FUNCTION_BLOCK FB 1001
TITLE = HOPPER
//Creation:
//Date:            Author:                                               Version
//-------------------------------------------------------------------------------
//-
//17.10.19          Ilia Bedniakov (ilia   )                             01.00.00
//
//Changes:
//No. Date:        Who       Description                           Mark   Version 
//-------------------------------------------------------------------------------
//- 
//               
//_______________________________________________________________________________
//_
//Function:
AUTHOR : ilia
NAME : project
VERSION : 0.1
VAR_INPUT
  i_xSystemActive : BOOL ;	//system control on
  i_xFAValveOpen : BOOL ;
  i_xFAValveClosed : BOOL ;
  i_xPBStart : BOOL ;	//Start Button
  i_xPBStop : BOOL ;	//StopButton
  i_xCstAvailable : BOOL ;	//Container On Place
  ack_FAValve : BOOL ;	//acknowlege FAValve
END_VAR
VAR_IN_OUT
  q_xFAValve : BOOL ;	//Open Fresh Air Valve
  q_xPFCMix : BOOL ;	//Container in position PFC to MIX01
  q_xLMStart : BOOL ;
  q_xLMCstAvalible : BOOL ;
  f_xFAValve : BOOL ;	//feedback fault
END_VAR
VAR
  reserve_IO : ARRAY  [4 .. 49 ] OF BYTE ;
  HMI : STRUCT 	//Interface of HMI
   CMD : STRUCT
    xxRes1 : BOOL ;
    xSetEmpty : BOOL ;
    xStopBtnTest : BOOL ;
    xStartBtnTest : BOOL ;
    xContainerPlaceTest : BOOL ;
    reserve_5 : BOOL ;
    reserve_6 : BOOL ;
    reserve_7 : BOOL ;
    reserve_8 : BOOL ;
    reserve_9 : BOOL ;
    reserve_10 : BOOL ;
    reserve_11 : BOOL ;
    reserve_12 : BOOL ;
    reserve_13 : BOOL ;
    reserve_14 : BOOL ;
    reserve_15 : BOOL ;
   END_STRUCT ;
   STATE : STRUCT
    xFaulted : BOOL ;
    xContainer : BOOL ;
    reserve_2 : BOOL ;
    reserve_3 : BOOL ;
    reserve_4 : BOOL ;
    xFilled : BOOL ;
    xEmpty : BOOL ;
    reserve_7 : BOOL ;
    reserve_8 : BOOL ;
    reserve_9 : BOOL ;
    reserve_10 : BOOL ;
    reserve_11 : BOOL ;
    reserve_12 : BOOL ;
    reserve_13 : BOOL ;
    reserve_14 : BOOL ;
    reserve_15 : BOOL ;
   END_STRUCT ;
   PARAM : STRUCT
    rDischargeTime : REAL  := 2.000000e+000;
    reserve_1 : REAL  := 6.000000e+001;
    reserve_2 : REAL  := 6.000000e+001;
    reserve_3 : REAL  := 6.000000e+001;
    reserve_4 : REAL ;
    reserve_5 : REAL ;
    reserve_6 : REAL ;
    reserve_7 : REAL ;
    reserve_8 : INT ;
    reserve_9 : INT ;
    reserve_10 : INT ;
    reserve_11 : INT ;
    reserve_12 : INT ;
    reserve_14 : INT ;
    reserve_15 : INT ;
   END_STRUCT ;
   PV : STRUCT
    rDischargeTime : REAL ;	//Minutes
    reserve_1_4 : REAL  := 6.000000e+001;
    reserve_2 : REAL  := 6.000000e+001;
    reserve_3 : REAL  := 6.000000e+001;
    reserve_4 : REAL ;
    reserve_5 : REAL ;
    reserve_6 : REAL ;
    reserve_7 : REAL ;
    iRecipeNumber : INT ;
    reserve_9 : INT ;
    reserve_10 : INT ;
    reserve_11 : INT ;
    reserve_12 : INT ;
    reserve_14 : INT ;
    reserve_15 : INT ;
   END_STRUCT ;
  END_STRUCT ;
  reserve_HMI : ARRAY  [146 .. 199 ] OF BYTE ;
  PROD : STRUCT 	//Interface of Production
   FROM : STRUCT
    reserve : INT ;
    reserve_1 : INT ;
    reserve_2 : INT ;
    reserve_3 : INT ;
    reserve_4 : INT ;
    reserve_5 : REAL ;
    reserve_6 : REAL ;
    CMD : STRUCT
     reserve : BOOL ;
     reserve_1 : BOOL ;
     reserve_2 : BOOL ;
     reserve_3 : BOOL ;
     reserve_4 : BOOL ;
     reserve_5 : BOOL ;
     reserve_6 : BOOL ;
     reserve_7 : BOOL ;
     reserve_8 : BOOL ;
     reserve_9 : BOOL ;
     reserve_10 : BOOL ;
     reserve_11 : BOOL ;
     reserve_12 : BOOL ;
     reserve_13 : BOOL ;
     reserve_14 : BOOL ;
     reserve_15 : BOOL ;
    END_STRUCT ;
   END_STRUCT ;
   TO : STRUCT
    reserve : INT ;
    reserve_1 : INT ;
    reserve_2 : INT ;
    reserve_3 : INT ;
    reserve_4 : INT ;
    reserve_5 : REAL ;
    reserve_6 : REAL ;
    STATE : STRUCT
     reserve : BOOL ;
     reserve_1 : BOOL ;
     reserve_2 : BOOL ;
     reserve_3 : BOOL ;
     reserve_4 : BOOL ;
     reserve_5 : BOOL ;
     reserve_6 : BOOL ;
     reserve_7 : BOOL ;
     reserve_8 : BOOL ;
     reserve_9 : BOOL ;
     reserve_10 : BOOL ;
     reserve_11 : BOOL ;
     reserve_12 : BOOL ;
     reserve_13 : BOOL ;
     reserve_14 : BOOL ;
     reserve_15 : BOOL ;
    END_STRUCT ;
   END_STRUCT ;
   reserve : ARRAY  [40 .. 49 ] OF BYTE ;
  END_STRUCT ;
  IF_CONSUMER : STRUCT 	//Interface scale in storage location
   CONTROL : STRUCT
    Answer_DB : INT ;
    Answer_DW : INT ;
    iRecipeNumber : INT ;
    rRes1 : REAL ;
    iPulseValve : REAL ;
    iPauseValve : REAL ;
    CMD : STRUCT
     xConnect : BOOL ;
     xRequest : BOOL ;
     xRelease : BOOL ;
     xFull : BOOL ;
     xCleaningRelease : BOOL ;
     xPressureFault : BOOL ;
     xAckRecipe : BOOL ;
     xPulseCondition : BOOL ;
     xDischargeActive : BOOL ;
     reserve_9 : BOOL ;
     reserve_10 : BOOL ;
     reserve_11 : BOOL ;
     reserve_12 : BOOL ;
     reserve_13 : BOOL ;
     reserve_14 : BOOL ;
     reserve_15 : BOOL ;
    END_STRUCT ;
   END_STRUCT ;
   STATUS : STRUCT
    reserve_1 : INT ;
    reserve_2 : INT ;
    iRecipeNumber : INT ;
    rRes1 : REAL ;
    rRes2 : REAL ;
    rRes3 : REAL ;
    STATE : STRUCT
     xReady : BOOL ;
     xActive : BOOL ;
     xStopped : BOOL ;
     xStarted : BOOL ;
     xEmpty : BOOL ;
     reserve_5 : BOOL ;
     reserve_6 : BOOL ;
     reserve_7 : BOOL ;
     reserve_8 : BOOL ;
     reserve_9 : BOOL ;
     reserve_10 : BOOL ;
     reserve_11 : BOOL ;
     reserve_12 : BOOL ;
     reserve_13 : BOOL ;
     reserve_14 : BOOL ;
     reserve_15 : BOOL ;
    END_STRUCT ;
   END_STRUCT ;
  END_STRUCT ;
  reserve_IF : ARRAY  [290 .. 499 ] OF BYTE ;
  FAValve : STRUCT 	//valve object with 1Q and 0-2I
   parameter : STRUCT
    valve_on : BOOL  := TRUE;	//activate valve structure
    clock_on : BOOL  := TRUE;	//activate clock structure
    reserve_3 : BOOL ;
    switching_number_on : BOOL ;	//activate switching number counter
    reserve_4 : BOOL ;
    parameter_1Q : BOOL ;	//valve type with 1 quit 0 inputs
    parameter_1Q_1I : BOOL ;	//valve type with 1 quit 1 input (=)
    parameter_1Q_1IN : BOOL ;	//valve type with 1 quit 1 input (<>)
    parameter_1Q_2I : BOOL  := TRUE;	//valve type with 1 quit 2 inputs
    parameter_text_pos_1 : BOOL ;
    parameter_text_straight : BOOL ;
    parameter_text_inverse : BOOL  := TRUE;	//select text inverse = "close/open" or "bypass/convey" aso.
    parameter_text_open : BOOL  := TRUE;	//select text quit = "open/close"
    parameter_text_convey : BOOL ;	//select text quit = "convey/bypass"
    parameter_text_on : BOOL ;	//select text quit = "on/off"
    parameter_text_up : BOOL ;	//select text quit = "up/down"
   END_STRUCT ;
   quit_valve : BOOL ;	//1 = quit valve
   input_valve_set : BOOL ;	//1 = input valve, if quit valve set
   input_valve_not_set : BOOL ;	//1 = input valve, if quit valve not set
   auto_mode_control : BOOL ;	//1 = release/control of valve in auto mode
   valve_in_operation : BOOL ;	//1 = signal valve in operation
   fault : BOOL ;	//1 = signal valve fault
   man_mode_to_SCADA : BOOL ;	//0 = automatic mode , 1 = manual mode
   man_mode_from_SCADA : BOOL ;	//0 = automatic mode , 1 = manual mode
   man_mode_control : BOOL ;	//1 = release/control of valve in manual mode (from SCADA)
   man_mode_locked : BOOL ;	//1 = change to manual mode locked, valve is in automatic use
   start_with_impulse : BOOL  := TRUE;	//1 = start cycle with impluse
   set_cycles_reached : BOOL ;	//1 = set number of cycles has been reached
   continous_clock : BOOL  := TRUE;	//1 = continous clock / 0 = set number of clocks
   simulation : BOOL ;	//1 = simulation of object
   release_clock : BOOL  := TRUE;	//1 = release bit for clock FC
   quit_clock : BOOL ;	//quit for clock FC, if release_clock = TRUE
   set_time_fault : INT  := 5;	//fault evaluation time in seconds
   actual_time_fault : INT ;	//actual fault evaluation time in seconds
   impulse_time : REAL  := 5.000000e+000;	//impulse time for clock in seconds
   break_time : REAL  := 5.000000e+000;	//break time for clock in seconds
   time_counter : REAL ;	//time counter (elapsed time)
   set_cycles : INT ;	//number of clocks if not continous clock
   clock_counter : INT ;	//clock counter
   switching_number_counter : STRUCT 	//switching number counter
    reset : BOOL ;	//reset switching number counter
    warning : BOOL ;	//warning number exceeded
    alarm : BOOL ;	//alarm number exceeded
    flank_flag : BOOL ;	//internal flag
    actual_switching_number : REAL ;	//actual switching number
    set_number_warning : REAL ;	//set number for warning
    set_number_alarm : REAL ;	//set number for alarm
   END_STRUCT ;
   set_time_in_operation : INT ;	//1IoO: set time for delay of "valve in operation"
   real_time_in_operation : INT ;	//1IoO: real time for delay of "valve in operation"
   system_on : BOOL ;	//system released resepectively system area released after emergency stopping
   reserve : ARRAY  [44 .. 47 ] OF BYTE ;
   object_state : INT ;	//1=grey; 5=green; 9=white; 15=yellow; 16=red
  END_STRUCT ;
  reserve_Cmod_1 : ARRAY  [550 .. 799 ] OF BYTE ;
  BinaryObjects : STRUCT
   PBStart : STRUCT
    parameter : STRUCT
     reserve : BOOL ;
     debounce_time : BOOL ;	//view/edit debounce time
     reserve_2 : BOOL ;
     switching_number_counter : BOOL ;	//Counter for operating cycles
     reserve_4 : BOOL ;
     reserve_5 : BOOL ;
     reserve_6 : BOOL ;
     reserve_7 : BOOL ;
     parameter_invers : BOOL ;	//Parameter signal invers, invert the status
     reserve_9 : BOOL ;
     reserve_10 : BOOL ;
     reserve_11 : BOOL ;
     reserve_12 : BOOL ;
     reserve_13 : BOOL ;
     reserve_14 : BOOL ;
     reserve_15 : BOOL ;
    END_STRUCT ;
    input_processed : BOOL ;	//Input_signal processed
    input : BOOL ;	//Input signal
    def_invert_input : BOOL ;	//Definition to invert input signal (1=invert input)
    def_debounce_input : BOOL ;	//Definition to debounce input signal (1=debounce input)
    def_fault_state : BOOL ;	//Definition of fault state
    fault : BOOL ;	//1 = fault message
    man_mode_to_SCADA : BOOL ;	//0=Automode; 1=Manualmode
    man_mode_from_SCADA : BOOL ;	//0=Automode; 1=Manualmode
    man_mode_control : BOOL ;	//Control the object in manual mode (from scada)
    man_mode_locked : BOOL ;	//Lock manual mode, because object is used in auto mode
    system_on : BOOL ;
    spare : BOOL ;
    input_inverted : BOOL ;	//Input signal inverted if necessary
    input_debounced : BOOL ;	//Input signal debounced if necessary (also inverted if necessary9)
    input_debounced_high : BOOL ;	//Input signal debounced high (output signal timer)
    input_debounced_low : BOOL ;	//Input signal debounced low (output signal timer)
    set_time_fault : INT ;	//Set value fault evaulation time
    act_time_fault : INT ;	//Act value fault avaulation time
    set_time_debounced_high : REAL ;
    act_time_debounced_high : REAL ;
    set_time_debounced_low : REAL ;
    act_time_debounced_low : REAL ;
    cycle_counter : STRUCT
     reset_counter : BOOL ;	//Reset operating cycle counter
     warning : BOOL ;	//Warning time 1 elapsed
     alarm : BOOL ;	//Alarm time 2 elapsed
     flank_flag : BOOL ;	//Intern used flag
     act_number_of_cycles : REAL ;	//Actual number of cycles (cycle counter)
     set_number_warning : REAL ;	//Set value for generate the warning
     set_number_alarm : REAL ;	//Set value for generate the alarm
    END_STRUCT ;
    reserve : ARRAY  [38 .. 47 ] OF BYTE ;
    object_state : INT ;
   END_STRUCT ;
   PBStop : STRUCT
    parameter : STRUCT
     reserve : BOOL ;
     debounce_time : BOOL ;	//view/edit debounce time
     reserve_2 : BOOL ;
     switching_number_counter : BOOL ;	//Counter for operating cycles
     reserve_4 : BOOL ;
     reserve_5 : BOOL ;
     reserve_6 : BOOL ;
     reserve_7 : BOOL ;
     parameter_invers : BOOL ;	//Parameter signal invers, invert the status
     reserve_9 : BOOL ;
     reserve_10 : BOOL ;
     reserve_11 : BOOL ;
     reserve_12 : BOOL ;
     reserve_13 : BOOL ;
     reserve_14 : BOOL ;
     reserve_15 : BOOL ;
    END_STRUCT ;
    input_processed : BOOL ;	//Input_signal processed
    input : BOOL ;	//Input signal
    def_invert_input : BOOL ;	//Definition to invert input signal (1=invert input)
    def_debounce_input : BOOL ;	//Definition to debounce input signal (1=debounce input)
    def_fault_state : BOOL ;	//Definition of fault state
    fault : BOOL ;	//1 = fault message
    man_mode_to_SCADA : BOOL ;	//0=Automode; 1=Manualmode
    man_mode_from_SCADA : BOOL ;	//0=Automode; 1=Manualmode
    man_mode_control : BOOL ;	//Control the object in manual mode (from scada)
    man_mode_locked : BOOL ;	//Lock manual mode, because object is used in auto mode
    system_on : BOOL ;
    spare : BOOL ;
    input_inverted : BOOL ;	//Input signal inverted if necessary
    input_debounced : BOOL ;	//Input signal debounced if necessary (also inverted if necessary9)
    input_debounced_high : BOOL ;	//Input signal debounced high (output signal timer)
    input_debounced_low : BOOL ;	//Input signal debounced low (output signal timer)
    set_time_fault : INT ;	//Set value fault evaulation time
    act_time_fault : INT ;	//Act value fault avaulation time
    set_time_debounced_high : REAL ;
    act_time_debounced_high : REAL ;
    set_time_debounced_low : REAL ;
    act_time_debounced_low : REAL ;
    cycle_counter : STRUCT
     reset_counter : BOOL ;	//Reset operating cycle counter
     warning : BOOL ;	//Warning time 1 elapsed
     alarm : BOOL ;	//Alarm time 2 elapsed
     flank_flag : BOOL ;	//Intern used flag
     act_number_of_cycles : REAL ;	//Actual number of cycles (cycle counter)
     set_number_warning : REAL ;	//Set value for generate the warning
     set_number_alarm : REAL ;	//Set value for generate the alarm
    END_STRUCT ;
    reserve : ARRAY  [38 .. 47 ] OF BYTE ;
    object_state : INT ;
   END_STRUCT ;
   PBCstAvailable : STRUCT
    parameter : STRUCT
     reserve : BOOL ;
     debounce_time : BOOL ;	//view/edit debounce time
     reserve_2 : BOOL ;
     switching_number_counter : BOOL ;	//Counter for operating cycles
     reserve_4 : BOOL ;
     reserve_5 : BOOL ;
     reserve_6 : BOOL ;
     reserve_7 : BOOL ;
     parameter_invers : BOOL ;	//Parameter signal invers, invert the status
     reserve_9 : BOOL ;
     reserve_10 : BOOL ;
     reserve_11 : BOOL ;
     reserve_12 : BOOL ;
     reserve_13 : BOOL ;
     reserve_14 : BOOL ;
     reserve_15 : BOOL ;
    END_STRUCT ;
    input_processed : BOOL ;	//Input_signal processed
    input : BOOL ;	//Input signal
    def_invert_input : BOOL ;	//Definition to invert input signal (1=invert input)
    def_debounce_input : BOOL ;	//Definition to debounce input signal (1=debounce input)
    def_fault_state : BOOL ;	//Definition of fault state
    fault : BOOL ;	//1 = fault message
    man_mode_to_SCADA : BOOL ;	//0=Automode; 1=Manualmode
    man_mode_from_SCADA : BOOL ;	//0=Automode; 1=Manualmode
    man_mode_control : BOOL ;	//Control the object in manual mode (from scada)
    man_mode_locked : BOOL ;	//Lock manual mode, because object is used in auto mode
    system_on : BOOL ;
    spare : BOOL ;
    input_inverted : BOOL ;	//Input signal inverted if necessary
    input_debounced : BOOL ;	//Input signal debounced if necessary (also inverted if necessary9)
    input_debounced_high : BOOL ;	//Input signal debounced high (output signal timer)
    input_debounced_low : BOOL ;	//Input signal debounced low (output signal timer)
    set_time_fault : INT ;	//Set value fault evaulation time
    act_time_fault : INT ;	//Act value fault avaulation time
    set_time_debounced_high : REAL ;
    act_time_debounced_high : REAL ;
    set_time_debounced_low : REAL ;
    act_time_debounced_low : REAL ;
    cycle_counter : STRUCT
     reset_counter : BOOL ;	//Reset operating cycle counter
     warning : BOOL ;	//Warning time 1 elapsed
     alarm : BOOL ;	//Alarm time 2 elapsed
     flank_flag : BOOL ;	//Intern used flag
     act_number_of_cycles : REAL ;	//Actual number of cycles (cycle counter)
     set_number_warning : REAL ;	//Set value for generate the warning
     set_number_alarm : REAL ;	//Set value for generate the alarm
    END_STRUCT ;
    reserve : ARRAY  [38 .. 47 ] OF BYTE ;
    object_state : INT ;
   END_STRUCT ;
  END_STRUCT ;
  reserve_Cmod : ARRAY  [950 .. 1499 ] OF BYTE ;
  TIMES : STRUCT 	//ten timers
   TON_VibroRinneFault : STRUCT
    IN : BOOL ;
    RST : BOOL ;
    IMP : BOOL ;
    Q : BOOL ;
    PT : REAL ;
    ET : REAL ;
   END_STRUCT ;
   TON_Restdischarge : STRUCT
    IN : BOOL ;
    RST : BOOL ;
    IMP : BOOL ;
    Q : BOOL ;
    PT : REAL ;
    ET : REAL ;
   END_STRUCT ;
   TON_VibroRinneStart : STRUCT
    IN : BOOL ;
    RST : BOOL ;
    IMP : BOOL ;
    Q : BOOL ;
    PT : REAL ;
    ET : REAL ;
   END_STRUCT ;
   TON_HopperDischarge : STRUCT
    IN : BOOL ;
    RST : BOOL ;
    IMP : BOOL ;
    Q : BOOL ;
    PT : REAL ;
    ET : REAL ;
   END_STRUCT ;
   TON_Vibrorinne : STRUCT
    IN : BOOL ;
    RST : BOOL ;
    IMP : BOOL ;
    Q : BOOL ;
    PT : REAL ;
    ET : REAL ;
   END_STRUCT ;
  END_STRUCT ;
  SEQUENCES : STRUCT
   Filling : STRUCT
    AUTO : BOOL ;
    MANUAL : BOOL ;
    LOCKED : BOOL ;
    reserve : BOOL ;
    reserve_1 : BOOL ;
    reserve_2 : BOOL ;
    reserve_3 : BOOL ;
    reserve_4 : BOOL ;
    reserve_5 : BOOL ;
    reserve_6 : BOOL ;
    reserve_7 : BOOL ;
    reserve_8 : BOOL ;
    reserve_9 : BOOL ;
    reserve_10 : BOOL ;
    reserve_11 : BOOL ;
    reserve_12 : BOOL ;
   END_STRUCT ;
   Discharging : STRUCT
    AUTO : BOOL ;
    MANUAL : BOOL ;
    LOCKED : BOOL ;
    RELEASED : BOOL ;
    ACTIVE : BOOL ;
    HOPPERDISCHARGE : BOOL ;
    FAULTED : BOOL ;
    CLEANING : BOOL ;
    reserve_5 : BOOL ;
    reserve_6 : BOOL ;
    reserve_7 : BOOL ;
    reserve_8 : BOOL ;
    reserve_9 : BOOL ;
    reserve_10 : BOOL ;
    reserve_11 : BOOL ;
    reserve_15 : BOOL ;
   END_STRUCT ;
   reserve : ARRAY  [4 .. 99 ] OF BYTE ;
  END_STRUCT ;
  INTERNAL : STRUCT
   IF : STRUCT
    RECEIVER : STRUCT
     res : BOOL ;
     res_1 : BOOL ;
     res_2 : BOOL ;
     res_3 : BOOL ;
     res_4 : BOOL ;
     res_5 : BOOL ;
     res_6 : BOOL ;
     res_7 : BOOL ;
    END_STRUCT ;
    reserve_1 : BOOL ;
    reserve_2 : BOOL ;
    reserve_3 : BOOL ;
    reserve_4 : BOOL ;
    reserve_5 : BOOL ;
    reserve_6 : BOOL ;
    reserve_7 : BOOL ;
    reserve_8 : BOOL ;
    reserve_9 : BOOL ;
    reserve_10 : BOOL ;
    reserve_11 : BOOL ;
    reserve_12 : BOOL ;
    reserve_13 : BOOL ;
    reserve_14 : BOOL ;
    reserve_14_1 : BOOL ;
   END_STRUCT ;
   Flags : STRUCT
    FP_start : STRUCT
     helpbit : BOOL ;
     pulsebit : BOOL ;
    END_STRUCT ;
    FN_cleaning : STRUCT
     helpbit : BOOL ;
     pulsebit : BOOL ;
    END_STRUCT ;
    res_2 : BOOL ;
    res_3 : BOOL ;
    res_2_1 : BOOL ;
    res_3_1 : BOOL ;
    res_3_1_1 : BOOL ;
   END_STRUCT ;
   CSTStatus : STRUCT
    xx_xFull : BOOL ;
    xFilled : BOOL ;
    xEmptyOrDischarged : BOOL ;
    xCSTAvailable : BOOL ;
    xCleanedPipe : BOOL ;
    reserve_5 : BOOL ;
    reserve_6 : BOOL ;
    reserve_7 : BOOL ;
    xValveExtraCond : BOOL ;
   END_STRUCT ;
   CSTProcessStatus : STRUCT
    xStartCMDActive : BOOL ;
    reserve_1 : BOOL ;
    reserve_2 : BOOL ;
    reserve_3 : BOOL ;
    reserve_4 : BOOL ;
    reserve_5 : BOOL ;
    reserve_6 : BOOL ;
    reserve_7 : BOOL ;
   END_STRUCT ;
   Switches : STRUCT
    res1 : BOOL ;
    res2 : BOOL ;
    res3 : BOOL ;
    res4 : BOOL ;
    res5 : BOOL ;
    res6 : BOOL ;
    res7 : BOOL ;
    ress8 : BOOL ;
    res9 : BOOL ;
    res10 : BOOL ;
    res11 : BOOL ;
   END_STRUCT ;
   BUTTONS_LAMPS : STRUCT
    LMStart : STRUCT
     Steady : BOOL ;
     Flash : BOOL ;
     DoubleFlash : BOOL ;
     Activated : BOOL ;
     res_1 : BOOL ;
     res_2 : BOOL ;
     res_3 : BOOL ;
     res_4 : BOOL ;
    END_STRUCT ;
    LMStop : STRUCT
     Steady : BOOL ;
     Flash : BOOL ;
     DoubleFlash : BOOL ;
     Activated : BOOL ;
     res_1 : BOOL ;
     res_2 : BOOL ;
     res_3 : BOOL ;
     res_4 : BOOL ;
    END_STRUCT ;
    LMCstAvailable : STRUCT
     Steady : BOOL ;
     Flash : BOOL ;
     DoubleFlash : BOOL ;
     Activated : BOOL ;
     res_1 : BOOL ;
     res_2 : BOOL ;
     res_3 : BOOL ;
     res_4 : BOOL ;
    END_STRUCT ;
    res_2_2 : BOOL ;
    res_3 : BOOL ;
    res_4 : BOOL ;
    res_5 : BOOL ;
    res_1_1 : BOOL ;
    res_2_1 : BOOL ;
    res_3_1 : BOOL ;
    res_4_1 : BOOL ;
    res_1 : BOOL ;
    res_2 : BOOL ;
   END_STRUCT ;
   Instance_DB_number : INT ;
  END_STRUCT ;
END_VAR
VAR_TEMP
  tempREAL : REAL ;
  tempINT : INT ;
  tempWORD : WORD ;
  tempBOOL : BOOL ;
END_VAR
BEGIN
NETWORK
TITLE = ------------------ INSTANCE DB (STANDART)-----------------------
      L     0;
      L     DINO;
      ==I;
      BEC;
      T     #INTERNAL.Instance_DB_number;
NETWORK
TITLE = -------------SEQUENCES AUTO/LOCKED/MANUAL-----------------
NETWORK
TITLE = Sequence discharging auto
      A     #IF_CONSUMER.CONTROL.CMD.xRequest;
      AN    #SEQUENCES.Discharging.LOCKED;
      =     #SEQUENCES.Discharging.AUTO;
NETWORK
TITLE = Sequence discharging manual
      O     #FAValve.man_mode_to_SCADA;
      =     #SEQUENCES.Discharging.MANUAL;
NETWORK
TITLE = Sequence discharging locked
      O     #SEQUENCES.Discharging.MANUAL;
      ON    #i_xSystemActive;
      =     #SEQUENCES.Discharging.LOCKED;
NETWORK
TITLE = ------------- SENSORS/SWITCHES/BINARY --------------------------
NETWORK
TITLE = LMP PBStart
      O     #i_xPBStart;
      O     #HMI.CMD.xStartBtnTest;
      =     #i_xPBStart;
      CALL  FC 24 (
           in_Handbedienung_erlaubt := TRUE,
           in_Anlage_ein            := #i_xSystemActive,
           in_Eingang               := #i_xPBStart,
           in_Eingang_drehen        := FALSE,
           in_Eingang_entprellen    := FALSE,
           in_Stoerauswertung_aktiv := FALSE,
           in_Quitt_Stoerung_noetig := FALSE,
           in_Stoer_Zustand         := FALSE,
           in_Quitt_Stoerung        := FALSE,
           io_Eingang_verarbeitet   := #INTERNAL.BUTTONS_LAMPS.LMStart.Activated,
           io_Stoerung              := #tempBOOL,
           io_Struktur              := #BinaryObjects.PBStart);
NETWORK
TITLE = PB STOP
      O     #i_xPBStop;
      O     #HMI.CMD.xStopBtnTest;
      =     #i_xPBStop;
      CALL  FC 24 (
           in_Handbedienung_erlaubt := TRUE,
           in_Anlage_ein            := #i_xSystemActive,
           in_Eingang               := #i_xPBStop,
           in_Eingang_drehen        := FALSE,
           in_Eingang_entprellen    := FALSE,
           in_Stoerauswertung_aktiv := FALSE,
           in_Quitt_Stoerung_noetig := FALSE,
           in_Stoer_Zustand         := FALSE,
           in_Quitt_Stoerung        := FALSE,
           io_Eingang_verarbeitet   := #INTERNAL.BUTTONS_LAMPS.LMStop.Activated,
           io_Stoerung              := #tempBOOL,
           io_Struktur              := #BinaryObjects.PBStop);
NETWORK
TITLE = Lmp PB CST Avalible
      O     #i_xCstAvailable;
      O     #HMI.CMD.xContainerPlaceTest;
      =     #i_xCstAvailable;
      CALL  FC 24 (
           in_Handbedienung_erlaubt := TRUE,
           in_Anlage_ein            := #i_xSystemActive,
           in_Eingang               := #i_xCstAvailable,
           in_Eingang_drehen        := FALSE,
           in_Eingang_entprellen    := FALSE,
           in_Stoerauswertung_aktiv := FALSE,
           in_Quitt_Stoerung_noetig := FALSE,
           in_Stoer_Zustand         := FALSE,
           in_Quitt_Stoerung        := FALSE,
           io_Eingang_verarbeitet   := #INTERNAL.BUTTONS_LAMPS.LMCstAvailable.Activated,
           io_Stoerung              := #tempBOOL,
           io_Struktur              := #BinaryObjects.PBCstAvailable);
NETWORK
TITLE = ------------SEQUENCES/HANDSHAKES DISCHARGING -----------
NETWORK
TITLE = Container available on position
      A     #INTERNAL.BUTTONS_LAMPS.LMCstAvailable.Activated;
      S     #INTERNAL.CSTStatus.xCSTAvailable;
      A     #IF_CONSUMER.CONTROL.CMD.xCleaningRelease;
      R     #INTERNAL.CSTStatus.xCSTAvailable;
NETWORK
TITLE = Number Recipe Internally
      A     #INTERNAL.CSTStatus.xCSTAvailable;
      JCN   TRC;
      L     #IF_CONSUMER.CONTROL.iRecipeNumber;
      T     #HMI.PV.iRecipeNumber;
TRC:  NOP   0;
NETWORK
TITLE = Start process internal command
//Discussion - with Start/Stop buttons or from Panel
      A     #i_xSystemActive;
      A     #INTERNAL.BUTTONS_LAMPS.LMStart.Activated;
      A     #IF_CONSUMER.CONTROL.CMD.xRequest;
      A     #INTERNAL.CSTStatus.xCSTAvailable;
      A     #SEQUENCES.Discharging.AUTO;
      FP    #INTERNAL.Flags.FP_start.helpbit;
      =     #INTERNAL.Flags.FP_start.pulsebit;
      A     #INTERNAL.Flags.FP_start.pulsebit;
      S     #INTERNAL.CSTProcessStatus.xStartCMDActive;
      ON    #i_xSystemActive;
      O     #i_xPBStop;
      O     #INTERNAL.BUTTONS_LAMPS.LMStop.Activated;
      R     #INTERNAL.CSTProcessStatus.xStartCMDActive;
NETWORK
TITLE = Discharging: FAULT SEQ
      O     #f_xFAValve;
      =     #SEQUENCES.Discharging.FAULTED;
NETWORK
TITLE = Discharging: RELEASE from REC01/ RELEASED SEQ
      A     #IF_CONSUMER.CONTROL.CMD.xRelease;
      A     #INTERNAL.CSTProcessStatus.xStartCMDActive;
      AN    #SEQUENCES.Discharging.CLEANING;
      =     #SEQUENCES.Discharging.RELEASED;
NETWORK
TITLE = Discharging: READY TO CONSUMER
      A     #SEQUENCES.Discharging.AUTO;
      A     #INTERNAL.CSTProcessStatus.xStartCMDActive;
      AN    #SEQUENCES.Discharging.FAULTED;
      =     #IF_CONSUMER.STATUS.STATE.xReady;
NETWORK
TITLE = Discharging: ACTIVE SEQ
      A     #SEQUENCES.Discharging.RELEASED;
      A     #FAValve.valve_in_operation;
      =     #SEQUENCES.Discharging.ACTIVE;
NETWORK
TITLE = Discharging: CLEANING SEQ
      A     #IF_CONSUMER.CONTROL.CMD.xCleaningRelease;
      AN    #SEQUENCES.Discharging.RELEASED;
      =     #SEQUENCES.Discharging.CLEANING;
      A     #SEQUENCES.Discharging.CLEANING;
      FN    #INTERNAL.Flags.FN_cleaning.helpbit;
      =     #INTERNAL.Flags.FN_cleaning.pulsebit;
      A     #INTERNAL.Flags.FN_cleaning.pulsebit;
      S     #INTERNAL.CSTStatus.xCleanedPipe;
      A     #SEQUENCES.Discharging.RELEASED;
      R     #INTERNAL.CSTStatus.xCleanedPipe;
NETWORK
TITLE = Discharging: ACTIVE TO CONSUMER
      A     #SEQUENCES.Discharging.ACTIVE;
      =     #IF_CONSUMER.STATUS.STATE.xActive;
NETWORK
TITLE = Discharging: Recipe exchange
      A     #IF_CONSUMER.CONTROL.CMD.xConnect;
      A(;
      L     #IF_CONSUMER.CONTROL.iRecipeNumber;
      L     #IF_CONSUMER.STATUS.iRecipeNumber;
      ==I;
      );
      O;
      A     #INTERNAL.CSTStatus.xEmptyOrDischarged;
      O;
      A     #IF_CONSUMER.CONTROL.CMD.xAckRecipe;
      JCN   LR;
      L     #IF_CONSUMER.CONTROL.iRecipeNumber;
LR:   T     #IF_CONSUMER.STATUS.iRecipeNumber;
NETWORK
TITLE = Discharging: Stop to REC
      AN    #INTERNAL.CSTProcessStatus.xStartCMDActive;
      A     #INTERNAL.BUTTONS_LAMPS.LMStop.Activated;
      =     #IF_CONSUMER.STATUS.STATE.xStopped;
NETWORK
TITLE = Discharging: Storage Recipe Back to Consumer
      L     #HMI.PV.iRecipeNumber;
      T     #IF_CONSUMER.STATUS.iRecipeNumber;
NETWORK
TITLE = --------------------HOPPER STATES-------------------------------
NETWORK
TITLE = CST statuses (empty_discharged/filled)
//filled
      A     #SEQUENCES.Discharging.RELEASED;
      S     #INTERNAL.CSTStatus.xFilled;
      A     #INTERNAL.CSTStatus.xCleanedPipe;
      R     #INTERNAL.CSTStatus.xFilled;
      AN    #INTERNAL.CSTStatus.xFilled;
      =     #INTERNAL.CSTStatus.xEmptyOrDischarged;
NETWORK
TITLE = CST to CONSUMER
      A     #INTERNAL.CSTStatus.xEmptyOrDischarged;
      =     #IF_CONSUMER.STATUS.STATE.xEmpty;
NETWORK
TITLE = ----------------RELEASES TO AGGREGATES-----------------------
NETWORK
TITLE = Discharging: Release Unload Valve
      A     #SEQUENCES.Discharging.RELEASED;
      O     #SEQUENCES.Discharging.CLEANING;
      L     #IF_CONSUMER.CONTROL.iPulseValve;
      T     #FAValve.impulse_time;
      L     #IF_CONSUMER.CONTROL.iPauseValve;
      T     #FAValve.break_time;
      A     #SEQUENCES.Discharging.RELEASED;
      =     #FAValve.auto_mode_control;
// man mode locked
      A     #FAValve.auto_mode_control;
      =     #FAValve.man_mode_locked;
      CALL  FC 21 (
           in_Ventil_Typ            := 1,
           in_Handbedienung_erlaubt := TRUE,
           in_Quitt_Stoerung_noetig := FALSE,
           in_Quitt_Stoerung        := #ack_FAValve,
           in_Anlage_ein            := #i_xSystemActive,
           in_Ansteuerung_Ventil    := #FAValve.auto_mode_control,
           in_Eingang_angesteuert   := #i_xFAValveOpen,
           in_Eingang_nicht_angest  := #i_xFAValveClosed,
           io_Ausgang_Ventil        := #q_xFAValve,
           io_Ventil_in_Betrieb     := #FAValve.valve_in_operation,
           io_Stoerung              := #FAValve.fault,
           io_Ventilstruktur        := #FAValve);
NETWORK
TITLE = -------------------STATUSES TO VISU-----------------------------
NETWORK
TITLE = ------------------------LAMPS-----------------------------------
NETWORK
TITLE = lamp PB Start
      A     #IF_CONSUMER.CONTROL.CMD.xRequest;
//    A     #INTERNAL.Flags.FHP_Statuses.HopperEmpty
      =     #INTERNAL.BUTTONS_LAMPS.LMStart.Flash;
      A     #SEQUENCES.Discharging.ACTIVE;
      AN    #SEQUENCES.Discharging.FAULTED;
      AN    #SEQUENCES.Discharging.CLEANING;
      =     #INTERNAL.BUTTONS_LAMPS.LMStart.Steady;
      A     #SEQUENCES.Discharging.CLEANING;
      =     #INTERNAL.BUTTONS_LAMPS.LMStart.DoubleFlash;
      CALL  FC 25 (
           Steady                   := #INTERNAL.BUTTONS_LAMPS.LMStart.Steady,
           Flash                    := #INTERNAL.BUTTONS_LAMPS.LMStart.Flash,
           DoubleFlash              := #INTERNAL.BUTTONS_LAMPS.LMStart.DoubleFlash,
           LampTest                 := M 9.7,
           Lamp                     := #q_xLMStart);
NETWORK
TITLE = lamp PB Cst Avalible
      A     #INTERNAL.CSTStatus.xCSTAvailable;
      =     #INTERNAL.BUTTONS_LAMPS.LMCstAvailable.Steady;
      AN    #INTERNAL.CSTStatus.xCSTAvailable;
      =     #INTERNAL.BUTTONS_LAMPS.LMCstAvailable.Flash;
      A     #IF_CONSUMER.CONTROL.CMD.xRequest;
      AN    #INTERNAL.CSTStatus.xCSTAvailable;
      =     #INTERNAL.BUTTONS_LAMPS.LMCstAvailable.DoubleFlash;
      CALL  FC 25 (
           Steady                   := #INTERNAL.BUTTONS_LAMPS.LMCstAvailable.Steady,
           Flash                    := #INTERNAL.BUTTONS_LAMPS.LMCstAvailable.Flash,
           DoubleFlash              := #INTERNAL.BUTTONS_LAMPS.LMCstAvailable.DoubleFlash,
           LampTest                 := M 9.7,
           Lamp                     := #q_xLMCstAvalible);
NETWORK
TITLE = ----------------------INTERFACES-------------------------------
NETWORK
TITLE = Receiver
      CALL  FC 41 (
           i_SST_von_Ziel           := #IF_CONSUMER.CONTROL,
           i_SST_an_Ziel            := #IF_CONSUMER.STATUS);
END_FUNCTION_BLOCK

FUNCTION_BLOCK FB 1011
TITLE = REC01
//Creation:
//Date:            Author:                                               Version
//--------------------------------------------------------------------------------
//14.04.2018     Ilia Bedniakov (ilia)                                   01.00.00
//
//Changes:
//No. Date:        Who       Description                           Mark   Version 
//--------------------------------------------------------------------------------
//01  12.01.2019  ilia       correction at comissioning            (001)  01.01.00
//
//
//_______________________________________________________________________________
//Function:
AUTHOR : ilia
NAME : project
VERSION : 0.1
VAR_INPUT
  I_iIFVacuumPumpDB : INT ;	//VacuumPump DB Nr
  I_iIFVacuumPumpDW : INT ;	//VacuumPump Interface Start DW Nr
  I_iIFStorageDB : INT ;
  I_iIFStorageDW : INT ;
  I_xSystemActive : BOOL ;	//system control on
  I_xAngleValveOpen : BOOL ;	//Angle Valve Close
  I_xAngleValveClose : BOOL ;	//Angle Valve Close
  i_xPendelFlapREC : BOOL ;	//Pendulum Flap
  i_xHighLevelREC : BOOL ;	//high level sensor
  I_xPFC_PM1 : BOOL ;	//PFC PM Hopper Big Components
  I_xPFC_PM2 : BOOL ;	//PFC PM Hopper Small Components
  i_xAckFullReceiver : BOOL ;
  i_xAckAngleValve : BOOL ;
END_VAR
VAR_IN_OUT
  q_xAngleValve : BOOL ;	//Angle Valve Open
  q_xCleaningValve : BOOL ;	//Filter Cleaning Valve
  q_xRepperValve : BOOL ;	//Rapper Valve
  q_xRedLamp : BOOL ;
  q_xYellowLamp : BOOL ;
  q_xGreenLamp : BOOL ;
  f_xAngleValve : BOOL ;	//Angle Valve Open
  f_xFullReceiver : BOOL ;	//Fault
  f_xNoStartConditions : BOOL ;
  f_xNoPFCRequest : BOOL ;
  fNotEnoughMaterial : BOOL ;
END_VAR
VAR
  reserve_IO : ARRAY  [12 .. 49 ] OF BYTE ;
  HMI : STRUCT 	//Interface of HMI
   CMD : STRUCT
    xRelease : BOOL  := TRUE;	//Start Recipe Btn
    xSetEmpty : BOOL ;	//VISU command button
    xAckDataSet : BOOL ;	//Ack Previous Recipe
    xResetRecipe : BOOL ;
    reserve_4 : BOOL ;
    reserve_5 : BOOL ;
    reserve_6 : BOOL ;
    reserve_7 : BOOL ;
    reserve_8 : BOOL ;
    reserve_9 : BOOL ;
    reserve_10 : BOOL ;
    reserve_11 : BOOL ;
    reserve_12 : BOOL ;
    reserve_13 : BOOL ;
    reserve_14 : BOOL ;
    reserve_15 : BOOL ;
   END_STRUCT ;
   STATE : STRUCT
    xChangeDataSetBlocked : BOOL ;
    xCleaningActive : BOOL ;
    xPFCRequestPM1 : BOOL ;
    xPFCRequestPM2 : BOOL ;
    xRecipeFalse : BOOL ;
    reserve_5 : BOOL ;
    xFault : BOOL ;
    xFull : BOOL ;
    xFilled : BOOL ;
    xEmpty : BOOL ;
    reserve_10 : BOOL ;
    reserve_11 : BOOL ;
    reserve_12 : BOOL ;
    reserve_13 : BOOL ;
    reserve_14 : BOOL ;
    reserve_15 : BOOL ;
   END_STRUCT ;
   PARAM : STRUCT
    rFillingTime : REAL  := 1.000000e+001;	//Off delay for screener time
    rCleaningTime : REAL  := 1.500000e+001;	//cleaning pipeline dutration
    rDischargingTime : REAL  := 3.000000e+001;	//after this time and not free LL sensor stop filling
    res_4 : REAL  := 1.000000e+001;	//Off delay for screener time
    res_4_1 : REAL  := 1.000000e+001;	//Off delay for screener time
    res_1_1 : REAL  := 3.000000e+001;	//after this time and not free LL sensor stop filling
    res_2 : REAL ;	//no new material + empty pressure -> warning
    res_3 : REAL  := 5.000000e+000;	//after enclosing HL sensor HP03 delay for discharg starts again
    iConvDataSet : INT  := 1;	//Set storage location HP01/HP02
    reserve_7 : INT ;
    reserve_8 : INT ;
    reserve_9 : INT ;
    reserve_10 : INT ;
    reserve_11 : INT ;
    res_6 : INT ;
   END_STRUCT ;
   PV : STRUCT
    rFillingTime : REAL  := 1.000000e+001;	//Off delay for screener time
    rCleaningTime : REAL  := 1.500000e+001;	//cleaning pipeline dutration
    rDischargingTime : REAL  := 3.000000e+001;	//after this time and not free LL sensor stop filling
    res_4 : REAL  := 1.000000e+001;	//Off delay for screener time
    res_4_1 : REAL  := 1.000000e+001;	//Off delay for screener time
    res_1_1 : REAL  := 3.000000e+001;	//after this time and not free LL sensor stop filling
    res_2 : REAL ;	//no new material + empty pressure -> warning
    res_3 : REAL  := 5.000000e+000;	//after enclosing HL sensor HP03 delay for discharg starts again
    iConvDataSet : INT  := 1;	//Set storage location HP01/HP02
    reserve_7 : INT ;
    reserve_8 : INT ;
    reserve_9 : INT ;
    reserve_10 : INT ;
    reserve_11 : INT ;
    res_6 : INT ;
   END_STRUCT ;
  END_STRUCT ;
  reserve_HMI : ARRAY  [146 .. 199 ] OF BYTE ;
  PROD : STRUCT 	//Interface of Production
   FROM : STRUCT
    reserve : INT ;
    reserve_1 : INT ;
    reserve_2 : INT ;
    reserve_3 : INT ;
    reserve_4 : INT ;
    reserve_5 : REAL ;
    reserve_6 : REAL ;
    CMD : STRUCT
     reserve : BOOL ;
     reserve_1 : BOOL ;
     reserve_2 : BOOL ;
     reserve_3 : BOOL ;
     reserve_4 : BOOL ;
     reserve_5 : BOOL ;
     reserve_6 : BOOL ;
     reserve_7 : BOOL ;
     reserve_8 : BOOL ;
     reserve_9 : BOOL ;
     reserve_10 : BOOL ;
     reserve_11 : BOOL ;
     reserve_12 : BOOL ;
     reserve_13 : BOOL ;
     reserve_14 : BOOL ;
     reserve_15 : BOOL ;
    END_STRUCT ;
   END_STRUCT ;
   TO : STRUCT
    reserve : INT ;
    reserve_1 : INT ;
    reserve_2 : INT ;
    reserve_3 : INT ;
    reserve_4 : INT ;
    reserve_5 : REAL ;
    reserve_6 : REAL ;
    STATE : STRUCT
     reserve : BOOL ;
     reserve_1 : BOOL ;
     reserve_2 : BOOL ;
     reserve_3 : BOOL ;
     reserve_4 : BOOL ;
     reserve_5 : BOOL ;
     reserve_6 : BOOL ;
     reserve_7 : BOOL ;
     reserve_8 : BOOL ;
     reserve_9 : BOOL ;
     reserve_10 : BOOL ;
     reserve_11 : BOOL ;
     reserve_12 : BOOL ;
     reserve_13 : BOOL ;
     reserve_14 : BOOL ;
     reserve_15 : BOOL ;
    END_STRUCT ;
   END_STRUCT ;
   reserve : ARRAY  [40 .. 49 ] OF BYTE ;
  END_STRUCT ;
  RecipeData : STRUCT
   iRecNumber : INT ;	//Recipe Data Set from HMI
   Recipe : STRUCT
    rSpeedVP01 : REAL  := 2.000000e+001;	//VP speed from Data Record
    rPauseTime : REAL  := 5.000000e+000;	//Unload valve Pause from Data Record
    rPulseTime : REAL  := 5.000000e+000;	//Unload valve Pulse from Data Record
    reserve : ARRAY  [12 .. 19 ] OF BYTE ;
   END_STRUCT ;
  END_STRUCT ;
  reserve_ProdRec : ARRAY  [272 .. 299 ] OF BYTE ;
  IF_VP : STRUCT 	//Interface Blower in active object
   STATUS : STRUCT
    reserve_1 : INT ;
    reserve_2 : INT ;
    reserve_3 : INT ;
    reserve_4 : INT ;
    reserve_5 : INT ;
    rActualPressure : REAL ;
    reserve_6 : REAL ;
    STATE : STRUCT
     xReady : BOOL ;
     xActive : BOOL ;
     xPressureFault : BOOL ;
     xEmptyPressure : BOOL ;
     xFault : BOOL ;
     reserve_2 : BOOL ;
     reserve_3 : BOOL ;
     reserve_4 : BOOL ;
     reserve_5 : BOOL ;
     reserve_6 : BOOL ;
     reserve_7 : BOOL ;
     reserve_8 : BOOL ;
     reserve_9 : BOOL ;
     reserve_10 : BOOL ;
     reserve_11 : BOOL ;
     reserve_12 : BOOL ;
    END_STRUCT ;
   END_STRUCT ;
   CONTROL : STRUCT
    Answer_DB : INT ;
    Answer_DW : INT ;
    SpeedVP : INT ;
    reserve_2 : INT ;
    reserve_3 : INT ;
    reserve_4 : REAL ;
    reserve_5 : REAL ;
    CMD : STRUCT
     xRequest : BOOL ;
     xRelease : BOOL ;
     reserve : BOOL ;
     reserve_1 : BOOL ;
     reserve_2 : BOOL ;
     reserve_3 : BOOL ;
     reserve_4 : BOOL ;
     reserve_5 : BOOL ;
     reserve_6 : BOOL ;
     reserve_7 : BOOL ;
     reserve_8 : BOOL ;
     reserve_9 : BOOL ;
     reserve_10 : BOOL ;
     reserve_11 : BOOL ;
     reserve_12 : BOOL ;
     reserve_13 : BOOL ;
    END_STRUCT ;
   END_STRUCT ;
  END_STRUCT ;
  IF_Storage : STRUCT
   STATUS : STRUCT
    iRes1 : INT ;
    iRes2 : INT ;
    iRecipeNumber : INT ;
    rRes1 : REAL ;
    rRes2 : REAL ;
    rRes3 : REAL ;
    STATE : STRUCT
     xReady : BOOL ;
     xActive : BOOL ;
     xStopped : BOOL ;
     xStarted : BOOL ;
     xEmpty : BOOL ;
     reserve_5 : BOOL ;
     reserve_6 : BOOL ;
     reserve_7 : BOOL ;
     reserve_8 : BOOL ;
     reserve_9 : BOOL ;
     reserve_10 : BOOL ;
     reserve_11 : BOOL ;
     reserve_12 : BOOL ;
     reserve_13 : BOOL ;
     reserve_14 : BOOL ;
     reserve_15 : BOOL ;
    END_STRUCT ;
   END_STRUCT ;
   CONTROL : STRUCT
    Answer_DB : INT ;
    Answer_DW : INT ;
    iRecipeNumber : INT ;
    rActualPressure : REAL ;
    iPulseValve : REAL ;
    iPauseValve : REAL ;
    CMD : STRUCT
     xConnect : BOOL ;
     xRequest : BOOL ;
     xRelease : BOOL ;
     xFull : BOOL ;
     xCleaningRelease : BOOL ;
     xPressureFault : BOOL ;
     xAckRecipe : BOOL ;
     res_2 : BOOL ;
     xDischargeActive : BOOL ;
     reserve_9 : BOOL ;
     reserve_10 : BOOL ;
     reserve_11 : BOOL ;
     reserve_12 : BOOL ;
     reserve_13 : BOOL ;
     reserve_14 : BOOL ;
     reserve_15 : BOOL ;
    END_STRUCT ;
   END_STRUCT ;
  END_STRUCT ;
  reserve_IF : ARRAY  [380 .. 499 ] OF BYTE ;
  AngleValve : STRUCT 	//Angle Valve 1Q 2I
   parameter : STRUCT
    valve_on : BOOL  := TRUE;	//activate valve structure
    clock_on : BOOL ;	//activate clock structure
    reserve_3 : BOOL ;
    switching_number_on : BOOL ;	//activate switching number counter
    reserve_4 : BOOL ;
    parameter_1Q : BOOL ;	//valve type with 1 quit 0 inputs
    parameter_1Q_1I : BOOL ;	//valve type with 1 quit 1 input (=)
    parameter_1Q_1IN : BOOL ;	//valve type with 1 quit 1 input (<>)
    parameter_1Q_2I : BOOL  := TRUE;	//valve type with 1 quit 2 inputs
    parameter_text_pos_1 : BOOL ;
    parameter_text_straight : BOOL ;
    parameter_text_inverse : BOOL ;	//select text inverse = "close/open" or "bypass/convey" aso.
    parameter_text_open : BOOL ;	//select text quit = "open/close"
    parameter_text_convey : BOOL  := TRUE;	//select text quit = "convey/bypass"
    parameter_text_on : BOOL ;	//select text quit = "on/off"
    parameter_text_up : BOOL ;	//select text quit = "up/down"
   END_STRUCT ;
   quit_valve : BOOL ;	//1 = quit valve
   input_valve_set : BOOL ;	//1 = input valve, if quit valve set
   input_valve_not_set : BOOL ;	//1 = input valve, if quit valve not set
   auto_mode_control : BOOL ;	//1 = release/control of valve in auto mode
   valve_in_operation : BOOL ;	//1 = signal valve in operation
   fault : BOOL ;	//1 = signal valve fault
   man_mode_to_SCADA : BOOL ;	//0 = automatic mode , 1 = manual mode
   man_mode_from_SCADA : BOOL ;	//0 = automatic mode , 1 = manual mode
   man_mode_control : BOOL ;	//1 = release/control of valve in manual mode (from SCADA)
   man_mode_locked : BOOL ;	//1 = change to manual mode locked, valve is in automatic use
   start_with_impulse : BOOL ;	//1 = start cycle with impluse
   set_cycles_reached : BOOL ;	//1 = set number of cycles has been reached
   continous_clock : BOOL ;	//1 = continous clock / 0 = set number of clocks
   simulation : BOOL ;	//1 = simulation of object
   release_clock : BOOL ;	//1 = release bit for clock FC
   quit_clock : BOOL ;	//quit for clock FC, if release_clock = TRUE
   set_time_fault : INT  := 5;	//fault evaluation time in seconds
   actual_time_fault : INT ;	//actual fault evaluation time in seconds
   impulse_time : REAL  := 5.000000e+000;	//impulse time for clock in seconds
   break_time : REAL  := 5.000000e+000;	//break time for clock in seconds
   time_counter : REAL ;	//time counter (elapsed time)
   set_cycles : INT ;	//number of clocks if not continous clock
   clock_counter : INT ;	//clock counter
   switching_number_counter : STRUCT 	//switching number counter
    reset : BOOL ;	//reset switching number counter
    warning : BOOL ;	//warning number exceeded
    alarm : BOOL ;	//alarm number exceeded
    flank_flag : BOOL ;	//internal flag
    actual_switching_number : REAL ;	//actual switching number
    set_number_warning : REAL ;	//set number for warning
    set_number_alarm : REAL ;	//set number for alarm
   END_STRUCT ;
   set_time_in_operation : INT ;	//1IoO: set time for delay of "valve in operation"
   real_time_in_operation : INT ;	//1IoO: real time for delay of "valve in operation"
   system_on : BOOL ;	//system released resepectively system area released after emergency stopping
   reserve : ARRAY  [44 .. 47 ] OF BYTE ;
   object_state : INT ;	//1=grey; 5=green; 9=white; 15=yellow; 16=red
  END_STRUCT ;
  FilterCleaning : STRUCT 	//Angle Valve 1Q 0I
   parameter : STRUCT
    valve_on : BOOL  := TRUE;	//activate valve structure
    clock_on : BOOL ;	//activate clock structure
    reserve_3 : BOOL ;
    switching_number_on : BOOL ;	//activate switching number counter
    reserve_4 : BOOL ;
    parameter_1Q : BOOL ;	//valve type with 1 quit 0 inputs
    parameter_1Q_1I : BOOL ;	//valve type with 1 quit 1 input (=)
    parameter_1Q_1IN : BOOL ;	//valve type with 1 quit 1 input (<>)
    parameter_1Q_2I : BOOL  := TRUE;	//valve type with 1 quit 2 inputs
    parameter_text_pos_1 : BOOL ;
    parameter_text_straight : BOOL ;
    parameter_text_inverse : BOOL ;	//select text inverse = "close/open" or "bypass/convey" aso.
    parameter_text_open : BOOL ;	//select text quit = "open/close"
    parameter_text_convey : BOOL  := TRUE;	//select text quit = "convey/bypass"
    parameter_text_on : BOOL ;	//select text quit = "on/off"
    parameter_text_up : BOOL ;	//select text quit = "up/down"
   END_STRUCT ;
   quit_valve : BOOL ;	//1 = quit valve
   input_valve_set : BOOL ;	//1 = input valve, if quit valve set
   input_valve_not_set : BOOL ;	//1 = input valve, if quit valve not set
   auto_mode_control : BOOL ;	//1 = release/control of valve in auto mode
   valve_in_operation : BOOL ;	//1 = signal valve in operation
   fault : BOOL ;	//1 = signal valve fault
   man_mode_to_SCADA : BOOL ;	//0 = automatic mode , 1 = manual mode
   man_mode_from_SCADA : BOOL ;	//0 = automatic mode , 1 = manual mode
   man_mode_control : BOOL ;	//1 = release/control of valve in manual mode (from SCADA)
   man_mode_locked : BOOL ;	//1 = change to manual mode locked, valve is in automatic use
   start_with_impulse : BOOL ;	//1 = start cycle with impluse
   set_cycles_reached : BOOL ;	//1 = set number of cycles has been reached
   continous_clock : BOOL ;	//1 = continous clock / 0 = set number of clocks
   simulation : BOOL ;	//1 = simulation of object
   release_clock : BOOL ;	//1 = release bit for clock FC
   quit_clock : BOOL ;	//quit for clock FC, if release_clock = TRUE
   set_time_fault : INT  := 5;	//fault evaluation time in seconds
   actual_time_fault : INT ;	//actual fault evaluation time in seconds
   impulse_time : REAL  := 5.000000e+000;	//impulse time for clock in seconds
   break_time : REAL  := 5.000000e+000;	//break time for clock in seconds
   time_counter : REAL ;	//time counter (elapsed time)
   set_cycles : INT ;	//number of clocks if not continous clock
   clock_counter : INT ;	//clock counter
   switching_number_counter : STRUCT 	//switching number counter
    reset : BOOL ;	//reset switching number counter
    warning : BOOL ;	//warning number exceeded
    alarm : BOOL ;	//alarm number exceeded
    flank_flag : BOOL ;	//internal flag
    actual_switching_number : REAL ;	//actual switching number
    set_number_warning : REAL ;	//set number for warning
    set_number_alarm : REAL ;	//set number for alarm
   END_STRUCT ;
   set_time_in_operation : INT ;	//1IoO: set time for delay of "valve in operation"
   real_time_in_operation : INT ;	//1IoO: real time for delay of "valve in operation"
   system_on : BOOL ;	//system released resepectively system area released after emergency stopping
   reserve : ARRAY  [44 .. 47 ] OF BYTE ;
   object_state : INT ;	//1=grey; 5=green; 9=white; 15=yellow; 16=red
  END_STRUCT ;
  Rapper : STRUCT 	//Angle Valve 1Q 0I
   parameter : STRUCT
    valve_on : BOOL  := TRUE;	//activate valve structure
    clock_on : BOOL ;	//activate clock structure
    reserve_3 : BOOL ;
    switching_number_on : BOOL ;	//activate switching number counter
    reserve_4 : BOOL ;
    parameter_1Q : BOOL ;	//valve type with 1 quit 0 inputs
    parameter_1Q_1I : BOOL ;	//valve type with 1 quit 1 input (=)
    parameter_1Q_1IN : BOOL ;	//valve type with 1 quit 1 input (<>)
    parameter_1Q_2I : BOOL  := TRUE;	//valve type with 1 quit 2 inputs
    parameter_text_pos_1 : BOOL ;
    parameter_text_straight : BOOL ;
    parameter_text_inverse : BOOL ;	//select text inverse = "close/open" or "bypass/convey" aso.
    parameter_text_open : BOOL ;	//select text quit = "open/close"
    parameter_text_convey : BOOL  := TRUE;	//select text quit = "convey/bypass"
    parameter_text_on : BOOL ;	//select text quit = "on/off"
    parameter_text_up : BOOL ;	//select text quit = "up/down"
   END_STRUCT ;
   quit_valve : BOOL ;	//1 = quit valve
   input_valve_set : BOOL ;	//1 = input valve, if quit valve set
   input_valve_not_set : BOOL ;	//1 = input valve, if quit valve not set
   auto_mode_control : BOOL ;	//1 = release/control of valve in auto mode
   valve_in_operation : BOOL ;	//1 = signal valve in operation
   fault : BOOL ;	//1 = signal valve fault
   man_mode_to_SCADA : BOOL ;	//0 = automatic mode , 1 = manual mode
   man_mode_from_SCADA : BOOL ;	//0 = automatic mode , 1 = manual mode
   man_mode_control : BOOL ;	//1 = release/control of valve in manual mode (from SCADA)
   man_mode_locked : BOOL ;	//1 = change to manual mode locked, valve is in automatic use
   start_with_impulse : BOOL ;	//1 = start cycle with impluse
   set_cycles_reached : BOOL ;	//1 = set number of cycles has been reached
   continous_clock : BOOL ;	//1 = continous clock / 0 = set number of clocks
   simulation : BOOL ;	//1 = simulation of object
   release_clock : BOOL ;	//1 = release bit for clock FC
   quit_clock : BOOL ;	//quit for clock FC, if release_clock = TRUE
   set_time_fault : INT  := 5;	//fault evaluation time in seconds
   actual_time_fault : INT ;	//actual fault evaluation time in seconds
   impulse_time : REAL  := 5.000000e+000;	//impulse time for clock in seconds
   break_time : REAL  := 5.000000e+000;	//break time for clock in seconds
   time_counter : REAL ;	//time counter (elapsed time)
   set_cycles : INT ;	//number of clocks if not continous clock
   clock_counter : INT ;	//clock counter
   switching_number_counter : STRUCT 	//switching number counter
    reset : BOOL ;	//reset switching number counter
    warning : BOOL ;	//warning number exceeded
    alarm : BOOL ;	//alarm number exceeded
    flank_flag : BOOL ;	//internal flag
    actual_switching_number : REAL ;	//actual switching number
    set_number_warning : REAL ;	//set number for warning
    set_number_alarm : REAL ;	//set number for alarm
   END_STRUCT ;
   set_time_in_operation : INT ;	//1IoO: set time for delay of "valve in operation"
   real_time_in_operation : INT ;	//1IoO: real time for delay of "valve in operation"
   system_on : BOOL ;	//system released resepectively system area released after emergency stopping
   reserve : ARRAY  [44 .. 47 ] OF BYTE ;
   object_state : INT ;	//1=grey; 5=green; 9=white; 15=yellow; 16=red
  END_STRUCT ;
  BinaryObjects : STRUCT
   PendulumFlap : STRUCT
    parameter : STRUCT
     reserve : BOOL ;
     debounce_time : BOOL  := TRUE;	//view/edit debounce time
     reserve_2 : BOOL  := TRUE;
     switching_number_counter : BOOL ;	//Counter for operating cycles
     reserve_4 : BOOL ;
     reserve_5 : BOOL ;
     reserve_6 : BOOL ;
     reserve_7 : BOOL ;
     parameter_invers : BOOL ;	//Parameter signal invers, invert the status
     reserve_9 : BOOL ;
     reserve_10 : BOOL ;
     reserve_11 : BOOL ;
     reserve_12 : BOOL ;
     reserve_13 : BOOL ;
     reserve_14 : BOOL ;
     reserve_15 : BOOL ;
    END_STRUCT ;
    input_processed : BOOL ;	//Input_signal processed
    input : BOOL ;	//Input signal
    def_invert_input : BOOL ;	//Definition to invert input signal (1=invert input)
    def_debounce_input : BOOL ;	//Definition to debounce input signal (1=debounce input)
    def_fault_state : BOOL ;	//Definition of fault state
    fault : BOOL ;	//1 = fault message
    man_mode_to_SCADA : BOOL ;	//0=Automode; 1=Manualmode
    man_mode_from_SCADA : BOOL ;	//0=Automode; 1=Manualmode
    man_mode_control : BOOL ;	//Control the object in manual mode (from scada)
    man_mode_locked : BOOL ;	//Lock manual mode, because object is used in auto mode
    system_on : BOOL ;
    spare : BOOL ;
    input_inverted : BOOL ;	//Input signal inverted if necessary
    input_debounced : BOOL ;	//Input signal debounced if necessary (also inverted if necessary9)
    input_debounced_high : BOOL ;	//Input signal debounced high (output signal timer)
    input_debounced_low : BOOL ;	//Input signal debounced low (output signal timer)
    set_time_fault : INT  := 5;	//Set value fault evaulation time
    act_time_fault : INT ;	//Act value fault avaulation time
    set_time_debounced_high : REAL ;
    act_time_debounced_high : REAL ;
    set_time_debounced_low : REAL ;
    act_time_debounced_low : REAL ;
    cycle_counter : STRUCT
     reset_counter : BOOL ;	//Reset operating cycle counter
     warning : BOOL ;	//Warning time 1 elapsed
     alarm : BOOL ;	//Alarm time 2 elapsed
     flank_flag : BOOL ;	//Intern used flag
     act_number_of_cycles : REAL ;	//Actual number of cycles (cycle counter)
     set_number_warning : REAL ;	//Set value for generate the warning
     set_number_alarm : REAL ;	//Set value for generate the alarm
    END_STRUCT ;
    reserve : ARRAY  [38 .. 47 ] OF BYTE ;
    object_state : INT ;
   END_STRUCT ;
   HighLevel : STRUCT
    parameter : STRUCT
     reserve : BOOL ;
     debounce_time : BOOL  := TRUE;	//view/edit debounce time
     reserve_2 : BOOL  := TRUE;
     switching_number_counter : BOOL ;	//Counter for operating cycles
     reserve_4 : BOOL ;
     reserve_5 : BOOL ;
     reserve_6 : BOOL ;
     reserve_7 : BOOL ;
     parameter_invers : BOOL ;	//Parameter signal invers, invert the status
     reserve_9 : BOOL ;
     reserve_10 : BOOL ;
     reserve_11 : BOOL ;
     reserve_12 : BOOL ;
     reserve_13 : BOOL ;
     reserve_14 : BOOL ;
     reserve_15 : BOOL ;
    END_STRUCT ;
    input_processed : BOOL ;	//Input_signal processed
    input : BOOL ;	//Input signal
    def_invert_input : BOOL ;	//Definition to invert input signal (1=invert input)
    def_debounce_input : BOOL ;	//Definition to debounce input signal (1=debounce input)
    def_fault_state : BOOL ;	//Definition of fault state
    fault : BOOL ;	//1 = fault message
    man_mode_to_SCADA : BOOL ;	//0=Automode; 1=Manualmode
    man_mode_from_SCADA : BOOL ;	//0=Automode; 1=Manualmode
    man_mode_control : BOOL ;	//Control the object in manual mode (from scada)
    man_mode_locked : BOOL ;	//Lock manual mode, because object is used in auto mode
    system_on : BOOL ;
    spare : BOOL ;
    input_inverted : BOOL ;	//Input signal inverted if necessary
    input_debounced : BOOL ;	//Input signal debounced if necessary (also inverted if necessary9)
    input_debounced_high : BOOL ;	//Input signal debounced high (output signal timer)
    input_debounced_low : BOOL ;	//Input signal debounced low (output signal timer)
    set_time_fault : INT  := 5;	//Set value fault evaulation time
    act_time_fault : INT ;	//Act value fault avaulation time
    set_time_debounced_high : REAL ;
    act_time_debounced_high : REAL ;
    set_time_debounced_low : REAL ;
    act_time_debounced_low : REAL ;
    cycle_counter : STRUCT
     reset_counter : BOOL ;	//Reset operating cycle counter
     warning : BOOL ;	//Warning time 1 elapsed
     alarm : BOOL ;	//Alarm time 2 elapsed
     flank_flag : BOOL ;	//Intern used flag
     act_number_of_cycles : REAL ;	//Actual number of cycles (cycle counter)
     set_number_warning : REAL ;	//Set value for generate the warning
     set_number_alarm : REAL ;	//Set value for generate the alarm
    END_STRUCT ;
    reserve : ARRAY  [38 .. 47 ] OF BYTE ;
    object_state : INT ;
   END_STRUCT ;
   PFC_PM1 : STRUCT
    parameter : STRUCT
     reserve : BOOL ;
     debounce_time : BOOL  := TRUE;	//view/edit debounce time
     reserve_2 : BOOL  := TRUE;
     switching_number_counter : BOOL ;	//Counter for operating cycles
     reserve_4 : BOOL ;
     reserve_5 : BOOL ;
     reserve_6 : BOOL ;
     reserve_7 : BOOL ;
     parameter_invers : BOOL ;	//Parameter signal invers, invert the status
     reserve_9 : BOOL ;
     reserve_10 : BOOL ;
     reserve_11 : BOOL ;
     reserve_12 : BOOL ;
     reserve_13 : BOOL ;
     reserve_14 : BOOL ;
     reserve_15 : BOOL ;
    END_STRUCT ;
    input_processed : BOOL ;	//Input_signal processed
    input : BOOL ;	//Input signal
    def_invert_input : BOOL ;	//Definition to invert input signal (1=invert input)
    def_debounce_input : BOOL ;	//Definition to debounce input signal (1=debounce input)
    def_fault_state : BOOL ;	//Definition of fault state
    fault : BOOL ;	//1 = fault message
    man_mode_to_SCADA : BOOL ;	//0=Automode; 1=Manualmode
    man_mode_from_SCADA : BOOL ;	//0=Automode; 1=Manualmode
    man_mode_control : BOOL ;	//Control the object in manual mode (from scada)
    man_mode_locked : BOOL ;	//Lock manual mode, because object is used in auto mode
    system_on : BOOL ;
    spare : BOOL ;
    input_inverted : BOOL ;	//Input signal inverted if necessary
    input_debounced : BOOL ;	//Input signal debounced if necessary (also inverted if necessary9)
    input_debounced_high : BOOL ;	//Input signal debounced high (output signal timer)
    input_debounced_low : BOOL ;	//Input signal debounced low (output signal timer)
    set_time_fault : INT  := 5;	//Set value fault evaulation time
    act_time_fault : INT ;	//Act value fault avaulation time
    set_time_debounced_high : REAL ;
    act_time_debounced_high : REAL ;
    set_time_debounced_low : REAL ;
    act_time_debounced_low : REAL ;
    cycle_counter : STRUCT
     reset_counter : BOOL ;	//Reset operating cycle counter
     warning : BOOL ;	//Warning time 1 elapsed
     alarm : BOOL ;	//Alarm time 2 elapsed
     flank_flag : BOOL ;	//Intern used flag
     act_number_of_cycles : REAL ;	//Actual number of cycles (cycle counter)
     set_number_warning : REAL ;	//Set value for generate the warning
     set_number_alarm : REAL ;	//Set value for generate the alarm
    END_STRUCT ;
    reserve : ARRAY  [38 .. 47 ] OF BYTE ;
    object_state : INT ;
   END_STRUCT ;
   PFC_PM2 : STRUCT
    parameter : STRUCT
     reserve : BOOL ;
     debounce_time : BOOL  := TRUE;	//view/edit debounce time
     reserve_2 : BOOL  := TRUE;
     switching_number_counter : BOOL ;	//Counter for operating cycles
     reserve_4 : BOOL ;
     reserve_5 : BOOL ;
     reserve_6 : BOOL ;
     reserve_7 : BOOL ;
     parameter_invers : BOOL ;	//Parameter signal invers, invert the status
     reserve_9 : BOOL ;
     reserve_10 : BOOL ;
     reserve_11 : BOOL ;
     reserve_12 : BOOL ;
     reserve_13 : BOOL ;
     reserve_14 : BOOL ;
     reserve_15 : BOOL ;
    END_STRUCT ;
    input_processed : BOOL ;	//Input_signal processed
    input : BOOL ;	//Input signal
    def_invert_input : BOOL ;	//Definition to invert input signal (1=invert input)
    def_debounce_input : BOOL ;	//Definition to debounce input signal (1=debounce input)
    def_fault_state : BOOL ;	//Definition of fault state
    fault : BOOL ;	//1 = fault message
    man_mode_to_SCADA : BOOL ;	//0=Automode; 1=Manualmode
    man_mode_from_SCADA : BOOL ;	//0=Automode; 1=Manualmode
    man_mode_control : BOOL ;	//Control the object in manual mode (from scada)
    man_mode_locked : BOOL ;	//Lock manual mode, because object is used in auto mode
    system_on : BOOL ;
    spare : BOOL ;
    input_inverted : BOOL ;	//Input signal inverted if necessary
    input_debounced : BOOL ;	//Input signal debounced if necessary (also inverted if necessary9)
    input_debounced_high : BOOL ;	//Input signal debounced high (output signal timer)
    input_debounced_low : BOOL ;	//Input signal debounced low (output signal timer)
    set_time_fault : INT  := 5;	//Set value fault evaulation time
    act_time_fault : INT ;	//Act value fault avaulation time
    set_time_debounced_high : REAL ;
    act_time_debounced_high : REAL ;
    set_time_debounced_low : REAL ;
    act_time_debounced_low : REAL ;
    cycle_counter : STRUCT
     reset_counter : BOOL ;	//Reset operating cycle counter
     warning : BOOL ;	//Warning time 1 elapsed
     alarm : BOOL ;	//Alarm time 2 elapsed
     flank_flag : BOOL ;	//Intern used flag
     act_number_of_cycles : REAL ;	//Actual number of cycles (cycle counter)
     set_number_warning : REAL ;	//Set value for generate the warning
     set_number_alarm : REAL ;	//Set value for generate the alarm
    END_STRUCT ;
    reserve : ARRAY  [38 .. 47 ] OF BYTE ;
    object_state : INT ;
   END_STRUCT ;
  END_STRUCT ;
  reserve_Cmod : ARRAY  [850 .. 949 ] OF BYTE ;
  TIMERS : STRUCT 	//ten timers
   TON_Cleaning : STRUCT
    IN : BOOL ;
    RST : BOOL ;
    IMP : BOOL ;
    Q : BOOL ;
    PT : REAL ;
    ET : REAL ;
   END_STRUCT ;
   TON_FillingTime : STRUCT
    IN : BOOL ;
    RST : BOOL ;
    IMP : BOOL ;
    Q : BOOL ;
    PT : REAL ;
    ET : REAL ;
   END_STRUCT ;
   TON_DischargingTime : STRUCT
    IN : BOOL ;
    RST : BOOL ;
    IMP : BOOL ;
    Q : BOOL ;
    PT : REAL ;
    ET : REAL ;
   END_STRUCT ;
   res_Timer_1 : STRUCT
    IN : BOOL ;
    RST : BOOL ;
    IMP : BOOL ;
    Q : BOOL ;
    PT : REAL ;
    ET : REAL ;
   END_STRUCT ;
   res_Timer_2 : STRUCT
    IN : BOOL ;
    RST : BOOL ;
    IMP : BOOL ;
    Q : BOOL ;
    PT : REAL ;
    ET : REAL ;
   END_STRUCT ;
   res_Timer_2_1 : STRUCT
    IN : BOOL ;
    RST : BOOL ;
    IMP : BOOL ;
    Q : BOOL ;
    PT : REAL ;
    ET : REAL ;
   END_STRUCT ;
  END_STRUCT ;
  SEQUENCES : STRUCT
   Filling : STRUCT
    AUTO : BOOL ;
    MANUAL : BOOL ;
    LOCKED : BOOL ;
    RELEASE : BOOL ;
    ACTIVE : BOOL ;
    CLEANING : BOOL ;
    FAULTED : BOOL ;
    reserve_4 : BOOL ;
    reserve_5 : BOOL ;
    reserve_6 : BOOL ;
    reserve_7 : BOOL ;
    reserve_8 : BOOL ;
    reserve_9 : BOOL ;
    reserve_10 : BOOL ;
    reserve_11 : BOOL ;
    reserve_12 : BOOL ;
   END_STRUCT ;
   Discharging : STRUCT
    AUTO : BOOL ;
    MANUAL : BOOL ;
    LOCKED : BOOL ;
    RELEASE : BOOL ;
    STAT1 : BOOL ;
    ACTIVE : BOOL ;
    res : BOOL ;
    reserve_1 : BOOL ;
    FAULTED : BOOL ;
    reserve_5 : BOOL ;
    reserve_6 : BOOL ;
    reserve_7 : BOOL ;
    reserve_8 : BOOL ;
    reserve_9 : BOOL ;
    reserve_10 : BOOL ;
    reserve_11 : BOOL ;
    reserve_12 : BOOL ;
   END_STRUCT ;
   reserve : ARRAY  [4 .. 99 ] OF BYTE ;
  END_STRUCT ;
  INTERNAL : STRUCT
   IF : STRUCT
    Storage : STRUCT
     StorageLocationNumber : INT ;
     StorageLocation_DB : INT ;
     StorageLocation_DW : INT ;
     reserve : INT ;
     res : BOOL ;
     IF_Silo_free : BOOL ;
     res_1 : BOOL ;
     res_2 : BOOL ;
     res_3 : BOOL ;
     res_4 : BOOL ;
     res_5 : BOOL ;
     res_6 : BOOL ;
    END_STRUCT ;
    Blower : STRUCT
     Blower_DB : INT ;
     Blower_DW : INT ;
     reserve : INT ;
     Blower_ready : BOOL ;
     Blower_free : BOOL ;
     reserve_2 : BOOL ;
     reserve_3 : BOOL ;
     reserve_1_1 : BOOL ;
     reserve_2_1 : BOOL ;
     reserve_3_1 : BOOL ;
     reserve_3_1_1 : BOOL ;
    END_STRUCT ;
    FC_RF : STRUCT
     RF_DB : INT ;
     RF_DW : INT ;
     reserve : INT ;
     RF_ready : BOOL ;
     RF_free : BOOL ;
     res : BOOL ;
     res_1 : BOOL ;
     res_2 : BOOL ;
     res_3 : BOOL ;
     res_4 : BOOL ;
     res_5 : BOOL ;
    END_STRUCT ;
    reserve_6 : BOOL ;
    reserve_7 : BOOL ;
    reserve_8 : BOOL ;
    reserve_9 : BOOL ;
    reserve_10 : BOOL ;
    reserve_11 : BOOL ;
    reserve_12 : BOOL ;
   END_STRUCT ;
   Flags : STRUCT
    FP_FalseDataset : STRUCT
     helpBit : BOOL ;
     pulseBit : BOOL ;
    END_STRUCT ;
    FP_CleaningRelease : STRUCT
     helpBit : BOOL ;
     pulseBit : BOOL ;
    END_STRUCT ;
    res_1 : BOOL ;
    res_2 : BOOL ;
    res_3 : BOOL ;
    res_4 : BOOL ;
    iCurrentRecipeNumber : INT ;
    iRes : BOOL ;
   END_STRUCT ;
   Switches : STRUCT
    xPendulumFlapClosed : BOOL ;
    xHighLevelCovered : BOOL ;
    xPM1Requested : BOOL ;
    xPM2Requested : BOOL ;
    res_3 : BOOL ;
    res_4 : BOOL ;
    res_5 : BOOL ;
    res_6 : BOOL ;
   END_STRUCT ;
   ReceiverStatus : STRUCT
    xFilled : BOOL ;
    xFull : BOOL ;
    xEmpty : BOOL ;
    res : BOOL ;
    res_1 : BOOL ;
    res_2 : BOOL ;
    res_3 : BOOL ;
    res_4 : BOOL ;
   END_STRUCT ;
   ProcessStatus : STRUCT
    xStoLocParTaken : BOOL ;
    xPipeCleaned : BOOL ;
    xStartRecipe : BOOL ;
    xRequestPM : BOOL ;
    res : BOOL ;
    res_1 : BOOL ;
    res_2 : BOOL ;
    res_3 : BOOL ;
   END_STRUCT ;
   BUTTONS_LAMPS : STRUCT
    LMStart : STRUCT
     Steady : BOOL ;
     Flash : BOOL ;
     DoubleFlash : BOOL ;
     Activated : BOOL ;
     res_1 : BOOL ;
     res_2 : BOOL ;
     res_3 : BOOL ;
     res_4 : BOOL ;
    END_STRUCT ;
    LMStop : STRUCT
     Steady : BOOL ;
     Flash : BOOL ;
     DoubleFlash : BOOL ;
     Activated : BOOL ;
     res_1 : BOOL ;
     res_2 : BOOL ;
     res_3 : BOOL ;
     res_4 : BOOL ;
    END_STRUCT ;
    Green : STRUCT
     Steady : BOOL ;
     Flash : BOOL ;
     DoubleFlash : BOOL ;
     res : BOOL ;
     res_1 : BOOL ;
     res_2 : BOOL ;
     res_3 : BOOL ;
     res_4 : BOOL ;
    END_STRUCT ;
    Yellow : STRUCT
     Steady : BOOL ;
     Flash : BOOL ;
     DoubleFlash : BOOL ;
     res : BOOL ;
     res_1 : BOOL ;
     res_2 : BOOL ;
     res_3 : BOOL ;
     res_4 : BOOL ;
    END_STRUCT ;
    Red : STRUCT
     Steady : BOOL ;
     Flash : BOOL ;
     DoubleFlash : BOOL ;
     res : BOOL ;
     res_1 : BOOL ;
     res_2 : BOOL ;
     res_3 : BOOL ;
     res_4 : BOOL ;
    END_STRUCT ;
    res_5 : BOOL ;
    res_1_1 : BOOL ;
    res_2_1 : BOOL ;
    res_3_1 : BOOL ;
    res_4_1 : BOOL ;
    res : BOOL ;
    res_1 : BOOL ;
    res_2 : BOOL ;
   END_STRUCT ;
   Instance_DB_number : INT ;
   Recipe : STRUCT
    iRecipeNumber : INT ;
    RecipeData : STRUCT 	//Recipe 1
     rSpeed : REAL ;	//VP speed from Data Record
     rPauseTime : REAL ;	//Unload valve Pause from Data Record
     rPulseTime : REAL ;	//Unload valve Pulse from Data Record
     reserve : ARRAY  [12 .. 19 ] OF BYTE ;
    END_STRUCT ;
   END_STRUCT ;
  END_STRUCT ;
END_VAR
VAR_TEMP
  StorageLoc_List_DW : INT ;
  StorageLocCopyError : INT ;
  tempDB : INT ;
  OffsetAddresse : INT ;
  outFault : INT ;
  dummyBOOL : BOOL ;
  silonumbertest : STRUCT
   silo1 : INT ;
   silo2 : INT ;
  END_STRUCT ;
END_VAR
BEGIN
NETWORK
TITLE = ------------------ INSTANCE DB (STANDART)-----------------------
      L     0;
      L     DINO;
      ==I;
      BEC;
      T     #INTERNAL.Instance_DB_number;
NETWORK
TITLE = ----------------SEQUENCES AUTO/LOCKED/MANUAL-----------------
NETWORK
TITLE = Sequence discharging auto
      AN    #SEQUENCES.Discharging.LOCKED;
      =     #SEQUENCES.Discharging.AUTO;
NETWORK
TITLE = Sequence discharging manual
//should be (ilia)
      CLR;
      =     #SEQUENCES.Discharging.MANUAL;
NETWORK
TITLE = Sequence discharging locked
      O     #SEQUENCES.Discharging.MANUAL;
      ON    #I_xSystemActive;
      =     #SEQUENCES.Discharging.LOCKED;
NETWORK
TITLE = Sequence filling auto
      AN    #SEQUENCES.Filling.LOCKED;
      =     #SEQUENCES.Filling.AUTO;
NETWORK
TITLE = Sequence filling manual
//manual = important motor is in manual, e.g. Rotary valve, screw, but in other 
//case CLR. Here angle valve is main part of unit
//AN    #SEQUENCES.Filling.AUTO
      O     #AngleValve.man_mode_to_SCADA;
      =     #SEQUENCES.Filling.MANUAL;
NETWORK
TITLE = Sequence filling locked
      AN    #I_xSystemActive;
      O     #SEQUENCES.Filling.MANUAL;
      =     #SEQUENCES.Filling.LOCKED;
NETWORK
TITLE = ---------------------SENSORS/SWITCHES --------------------------
NETWORK
TITLE = Pendulum Flap REC01
      CALL  FC 24 (
           in_Handbedienung_erlaubt := TRUE,
           in_Anlage_ein            := #I_xSystemActive,
           in_Eingang               := #i_xPendelFlapREC,
           in_Eingang_drehen        := FALSE,
           in_Eingang_entprellen    := TRUE,
           in_Stoerauswertung_aktiv := FALSE,
           in_Quitt_Stoerung_noetig := FALSE,
           in_Stoer_Zustand         := FALSE,
           in_Quitt_Stoerung        := FALSE,
           io_Eingang_verarbeitet   := #INTERNAL.Switches.xPendulumFlapClosed,
           io_Stoerung              := #BinaryObjects.PendulumFlap.fault,
           io_Struktur              := #BinaryObjects.PendulumFlap);	// close is close / no needed faultys
NETWORK
TITLE = High Level Sensor REC01
      CALL  FC 24 (
           in_Handbedienung_erlaubt := TRUE,
           in_Anlage_ein            := #I_xSystemActive,
           in_Eingang               := #i_xHighLevelREC,
           in_Eingang_drehen        := TRUE,
           in_Eingang_entprellen    := TRUE,
           in_Stoerauswertung_aktiv := TRUE,
           in_Quitt_Stoerung_noetig := TRUE,
           in_Stoer_Zustand         := FALSE,
           in_Quitt_Stoerung        := #i_xAckFullReceiver,
           io_Eingang_verarbeitet   := #INTERNAL.Switches.xHighLevelCovered,
           io_Stoerung              := #f_xFullReceiver,
           io_Struktur              := #BinaryObjects.HighLevel);
NETWORK
TITLE = PFC PM 1
      CALL  FC 24 (
           in_Handbedienung_erlaubt := TRUE,
           in_Anlage_ein            := #I_xSystemActive,
           in_Eingang               := #I_xPFC_PM1,
           in_Eingang_drehen        := FALSE,
           in_Eingang_entprellen    := TRUE,
           in_Stoerauswertung_aktiv := TRUE,
           in_Quitt_Stoerung_noetig := FALSE,
           in_Stoer_Zustand         := FALSE,
           in_Quitt_Stoerung        := TRUE,
           io_Eingang_verarbeitet   := #INTERNAL.Switches.xPM1Requested,
           io_Stoerung              := #BinaryObjects.PFC_PM1.fault,
           io_Struktur              := #BinaryObjects.PFC_PM1);
NETWORK
TITLE = PFC PM 2
      CALL  FC 24 (
           in_Handbedienung_erlaubt := TRUE,
           in_Anlage_ein            := #I_xSystemActive,
           in_Eingang               := #I_xPFC_PM2,
           in_Eingang_drehen        := FALSE,
           in_Eingang_entprellen    := TRUE,
           in_Stoerauswertung_aktiv := TRUE,
           in_Quitt_Stoerung_noetig := FALSE,
           in_Stoer_Zustand         := FALSE,
           in_Quitt_Stoerung        := TRUE,
           io_Eingang_verarbeitet   := #INTERNAL.Switches.xPM2Requested,
           io_Stoerung              := #BinaryObjects.PFC_PM2.fault,
           io_Struktur              := #BinaryObjects.PFC_PM2);
NETWORK
TITLE = -----------------------INPUT  PFC ------------------------------
NETWORK
TITLE = Discharging: Internal Request from PM
      O     #INTERNAL.Switches.xPM1Requested;
      O     #INTERNAL.Switches.xPM2Requested;
      =     #INTERNAL.ProcessStatus.xRequestPM;
NETWORK
TITLE = ----------------START NEW RECIPE------------------------------
NETWORK
TITLE = False Recipe number (Conveying Parameters)
//recipe =0
//OR
//new recipe AND REC NOT empty
//OR
//recipeREC <> REC CST
      A(;
      L     #RecipeData.iRecNumber;
      L     0;
      ==I;
      );
      O;
      A(;
      L     #RecipeData.iRecNumber;
      L     #IF_Storage.STATUS.iRecipeNumber;
      <>I;
      );
      A(;
      ON    #INTERNAL.ReceiverStatus.xEmpty;
      ON    #IF_Storage.STATUS.STATE.xEmpty;
      );
      S     #HMI.STATE.xRecipeFalse;
      A     #HMI.CMD.xAckDataSet;
      A(;
      L     #RecipeData.iRecNumber;
      L     #IF_Storage.STATUS.iRecipeNumber;
      ==I;
      );
      O     #HMI.CMD.xResetRecipe;
      R     #HMI.STATE.xRecipeFalse;
NETWORK
TITLE = Send Recipe to CST01
      A     #IF_Storage.STATUS.STATE.xEmpty;
      A(;
      L     #IF_Storage.STATUS.iRecipeNumber;
      L     #RecipeData.iRecNumber;
      <>I;
      );
      JCN   SRS;	// send recipe storage 
      T     #IF_Storage.CONTROL.iRecipeNumber;
SRS:  NOP   0;
NETWORK
TITLE = Start Recipe
      A     #HMI.CMD.xRelease;
      AN    #HMI.STATE.xRecipeFalse;
//     A     #INTERNAL.ReceiverStatus.xEmpty
//      O     
//      A(    
//      L     #INTERNAL.Flags.iCurrentRecipeNumber
//      L     #IF_Storage.STATUS.iRecipeNumber
//      ==I   
//      )     
      S     #INTERNAL.ProcessStatus.xStartRecipe;
      A(;
      L     #RecipeData.iRecNumber;
      L     #IF_Storage.STATUS.iRecipeNumber;
      <>I;
      );
      R     #INTERNAL.ProcessStatus.xStartRecipe;
//TODO TO LOOK
//     R     #INTERNAL.ProcessStatus.xStoLocParTaken
NETWORK
TITLE = Actual Recipe REC01
//New Data set - > Current Recipe
      A     #INTERNAL.ProcessStatus.xStartRecipe;
      FP    #INTERNAL.Flags.FP_FalseDataset.helpBit;
      JCN   WRA;	//write Recipe
      L     #RecipeData.iRecNumber;
      T     #INTERNAL.Flags.iCurrentRecipeNumber;
WRA:  NOP   0;
NETWORK
TITLE = Wrong start sequence - FAULT
      ON    #I_xSystemActive;
      O     #HMI.STATE.xRecipeFalse;
      O;
      A     #INTERNAL.ProcessStatus.xStartRecipe;
      A     #IF_Storage.CONTROL.CMD.xRequest;
      AN    #IF_Storage.STATUS.STATE.xReady;
      O;
      AN    #INTERNAL.ReceiverStatus.xEmpty;
      =     #f_xNoStartConditions;
NETWORK
TITLE = Block HMI Button for new Recipe 
      O     #SEQUENCES.Filling.ACTIVE;
      O     #SEQUENCES.Discharging.ACTIVE;
      =     #HMI.STATE.xChangeDataSetBlocked;
NETWORK
TITLE = Take Storage Location
      A     #INTERNAL.ProcessStatus.xStartRecipe;
      AN    #INTERNAL.ProcessStatus.xStoLocParTaken;
      JCN   SLT;	// storage location take
      A     #INTERNAL.ProcessStatus.xStartRecipe;
      =     #INTERNAL.ProcessStatus.xStoLocParTaken;
      L     #INTERNAL.Flags.iCurrentRecipeNumber;
      T     #HMI.PV.iConvDataSet;
SLT:  NOP   0;
NETWORK
TITLE = -------------SEQUENCES/HANDSHAKES FILLING --------------------
NETWORK
TITLE = Filling: Request to CST01
      A     #SEQUENCES.Filling.AUTO;
      A     #INTERNAL.ProcessStatus.xStartRecipe;
      =     #IF_Storage.CONTROL.CMD.xRequest;
NETWORK
TITLE = Filling: RELEASE SEQ
      A     #SEQUENCES.Filling.AUTO;
      A     #IF_Storage.CONTROL.CMD.xRequest;
      A     #IF_Storage.STATUS.STATE.xReady;
      AN    #SEQUENCES.Discharging.RELEASE;
      AN    #SEQUENCES.Filling.CLEANING;
      AN    #INTERNAL.ReceiverStatus.xFull;
      S     #SEQUENCES.Filling.RELEASE;
      A     #SEQUENCES.Discharging.RELEASE;
      O     #INTERNAL.ReceiverStatus.xFull;
      O     #TIMERS.TON_FillingTime.Q;
//    O     #IF_Storage.STATUS.STATE.xStopped
      ON    #IF_Storage.STATUS.STATE.xReady;
      R     #SEQUENCES.Filling.RELEASE;
NETWORK
TITLE = Filling: Filling Time
      A     #SEQUENCES.Filling.RELEASE;
      =     #TIMERS.TON_FillingTime.IN;
      CALL  FC 3 (
           in_Freigabe              := #TIMERS.TON_FillingTime.IN,
           in_Reset                 := #TIMERS.TON_FillingTime.RST,
           in_Impuls                := M 1.7,
           in_Impulszeit_in_100ms   := MW 6,
           in_Verzoegerungsart      := B#16#45,
           in_Verzoegerungszeit     := #HMI.PARAM.rFillingTime,
           io_Ausgangssignal        := #TIMERS.TON_FillingTime.Q,
           io_Zeitzaehler           := #TIMERS.TON_FillingTime.ET);
NETWORK
TITLE = Filling: CLEANING SEQ (Pipe cleaned BIT)
//Cleaned Reset
      A     #IF_Storage.STATUS.STATE.xActive;
      R     #INTERNAL.ProcessStatus.xPipeCleaned;
      A     #INTERNAL.ProcessStatus.xPipeCleaned;
      R     #SEQUENCES.Filling.CLEANING;
      A     #IF_Storage.STATUS.STATE.xStopped;
      AN    #INTERNAL.ProcessStatus.xPipeCleaned;
      A     #INTERNAL.ProcessStatus.xStartRecipe;
      FP    #INTERNAL.Flags.FP_CleaningRelease.helpBit;
      =     #INTERNAL.Flags.FP_CleaningRelease.pulseBit;
      A     #INTERNAL.Flags.FP_CleaningRelease.pulseBit;
      S     #SEQUENCES.Filling.CLEANING;
// Timer for sequence
      A     #SEQUENCES.Filling.CLEANING;
      =     #TIMERS.TON_Cleaning.IN;
      ON    #I_xSystemActive;
      =     #TIMERS.TON_Cleaning.RST;
      CALL  FC 3 (
           in_Freigabe              := #TIMERS.TON_Cleaning.IN,
           in_Reset                 := #TIMERS.TON_Cleaning.RST,
           in_Impuls                := M 1.7,
           in_Impulszeit_in_100ms   := MW 6,
           in_Verzoegerungsart      := B#16#45,
           in_Verzoegerungszeit     := #HMI.PARAM.rCleaningTime,
           io_Ausgangssignal        := #TIMERS.TON_Cleaning.Q,
           io_Zeitzaehler           := #TIMERS.TON_Cleaning.ET);
// right time to the HMI
      A     #TIMERS.TON_Cleaning.IN;
      AN    #TIMERS.TON_Cleaning.Q;
      L     0.000000e+00;
      JCN   RTH2;	//right time to HMI 
      L     #TIMERS.TON_Cleaning.ET;
RTH2: T     #HMI.PV.rCleaningTime;
// set help Bit
      A     #TIMERS.TON_Cleaning.Q;
      S     #INTERNAL.ProcessStatus.xPipeCleaned;
NETWORK
TITLE = Filling: Request BLOWER IF
      O     #SEQUENCES.Filling.RELEASE;
      O     #SEQUENCES.Filling.CLEANING;
      =     #IF_VP.CONTROL.CMD.xRequest;
NETWORK
TITLE = Filling: Frequency to BLOWER IF
      A     #IF_VP.CONTROL.CMD.xRequest;
      A     #IF_VP.STATUS.STATE.xReady;
      JCN   NBR;	// no request
      L     #RecipeData.Recipe.rSpeedVP01;
      T     #IF_VP.CONTROL.SpeedVP;
NBR:  NOP   0;
NETWORK
TITLE = Filling: Release BLOWER IF 
      A(;
      O     #SEQUENCES.Filling.RELEASE;
      O     #SEQUENCES.Filling.CLEANING;
      );
      A     #IF_VP.CONTROL.CMD.xRequest;
      A     #IF_VP.STATUS.STATE.xReady;
      =     #IF_VP.CONTROL.CMD.xRelease;
NETWORK
TITLE = Filling: Release STORAGE IF
//the condition about HP full has to be checked - may be it is necessary
      A     #SEQUENCES.Filling.RELEASE;
      A     #IF_Storage.CONTROL.CMD.xRequest;
      A     #IF_Storage.STATUS.STATE.xReady;
      A     #IF_VP.STATUS.STATE.xActive;
      AN    #IF_VP.STATUS.STATE.xPressureFault;
      A     #INTERNAL.ProcessStatus.xStoLocParTaken;
      AN    #IF_VP.STATUS.STATE.xPressureFault;
      =     #IF_Storage.CONTROL.CMD.xRelease;
NETWORK
TITLE = Filling: Actual Pressure to STORAGE IF
      L     #IF_VP.STATUS.rActualPressure;
      T     #IF_Storage.CONTROL.rActualPressure;
NETWORK
TITLE = Filling: Cleaning to STORAGE IF
      A     #SEQUENCES.Filling.CLEANING;
      =     #IF_Storage.CONTROL.CMD.xCleaningRelease;
NETWORK
TITLE = Filling: FAULTED SEQ
      O     #IF_VP.STATUS.STATE.xPressureFault;
      O     #IF_VP.STATUS.STATE.xFault;
      =     #SEQUENCES.Filling.FAULTED;
NETWORK
TITLE = Filling: ACTIVE SEQ
      A(;
      O     #SEQUENCES.Filling.RELEASE;
      O     #SEQUENCES.Filling.CLEANING;
      );
      A     #IF_VP.STATUS.STATE.xActive;
      A     #IF_Storage.STATUS.STATE.xActive;
      =     #SEQUENCES.Filling.ACTIVE;
NETWORK
TITLE = -------------SEQUENCES/HANDSHAKES DISCHARGING ------------
NETWORK
TITLE = Discharging: Discharging SEQ RELEASE (with timer)
      A     #SEQUENCES.Discharging.AUTO;
      A     #I_xSystemActive;
// A     #INTERNAL.ReceiverStatus.xFilled
      AN    #SEQUENCES.Filling.RELEASE;
      AN    #SEQUENCES.Filling.CLEANING;
      S     #SEQUENCES.Discharging.RELEASE;
      A     #SEQUENCES.Discharging.RELEASE;
      =     #TIMERS.TON_DischargingTime.IN;
      CALL  FC 3 (
           in_Freigabe              := #TIMERS.TON_DischargingTime.IN,
           in_Reset                 := #TIMERS.TON_DischargingTime.RST,
           in_Impuls                := M 1.7,
           in_Impulszeit_in_100ms   := MW 6,
           in_Verzoegerungsart      := B#16#45,
           in_Verzoegerungszeit     := #HMI.PARAM.rDischargingTime,
           io_Ausgangssignal        := #TIMERS.TON_DischargingTime.Q,
           io_Zeitzaehler           := #TIMERS.TON_DischargingTime.ET);
      A     #TIMERS.TON_DischargingTime.Q;
      A     #INTERNAL.ReceiverStatus.xEmpty;
      R     #SEQUENCES.Discharging.RELEASE;
// Timer to HMI
NETWORK
TITLE = Discharging: DISCHARGING ACTIVE
      A     #SEQUENCES.Discharging.AUTO;
      A     #SEQUENCES.Discharging.RELEASE;
      A     #INTERNAL.ProcessStatus.xRequestPM;
      =     #SEQUENCES.Discharging.ACTIVE;
      A     #SEQUENCES.Discharging.ACTIVE;
      =     #IF_Storage.CONTROL.CMD.xDischargeActive;
NETWORK
TITLE = -------------AGGREGATES ------------
NETWORK
TITLE = Filling: Angle Valve
      A     #SEQUENCES.Filling.RELEASE;
      O     #SEQUENCES.Filling.CLEANING;
      A     #IF_VP.CONTROL.CMD.xRelease;
      A     #IF_VP.STATUS.STATE.xActive;
      =     #AngleValve.auto_mode_control;
      A     #AngleValve.auto_mode_control;
      =     #AngleValve.man_mode_locked;
      CALL  FC 21 (
           in_Ventil_Typ            := 1,
           in_Handbedienung_erlaubt := M 11.0,
           in_Quitt_Stoerung_noetig := M 11.1,
           in_Quitt_Stoerung        := #i_xAckAngleValve,
           in_Anlage_ein            := #I_xSystemActive,
           in_Ansteuerung_Ventil    := #AngleValve.auto_mode_control,
           in_Eingang_angesteuert   := #I_xAngleValveOpen,
           in_Eingang_nicht_angest  := #I_xAngleValveClose,
           io_Ausgang_Ventil        := #q_xAngleValve,
           io_Ventil_in_Betrieb     := #AngleValve.valve_in_operation,
           io_Stoerung              := #AngleValve.fault,
           io_Ventilstruktur        := #AngleValve);
NETWORK
TITLE = Filling/Discharging: FilterCleaning Valve
      A     #SEQUENCES.Filling.RELEASE;
      O     #SEQUENCES.Filling.CLEANING;
      A     #IF_VP.CONTROL.CMD.xRelease;
      A     #IF_VP.STATUS.STATE.xActive;
      =     #FilterCleaning.auto_mode_control;
// man mode locked
      A     #FilterCleaning.auto_mode_control;
      AN    M 9.5;
      =     #FilterCleaning.man_mode_locked;
      CALL  FC 21 (
           in_Ventil_Typ            := 0,
           in_Handbedienung_erlaubt := TRUE,
           in_Quitt_Stoerung_noetig := FALSE,
           in_Quitt_Stoerung        := TRUE,
           in_Anlage_ein            := #I_xSystemActive,
           in_Ansteuerung_Ventil    := #FilterCleaning.auto_mode_control,
           in_Eingang_angesteuert   := FALSE,
           in_Eingang_nicht_angest  := FALSE,
           io_Ausgang_Ventil        := #q_xCleaningValve,
           io_Ventil_in_Betrieb     := #FilterCleaning.valve_in_operation,
           io_Stoerung              := #FilterCleaning.fault,
           io_Ventilstruktur        := #FilterCleaning);
NETWORK
TITLE = Discharging: RapperValve
      A     #SEQUENCES.Discharging.RELEASE;
      =     #Rapper.auto_mode_control;
// man mode locked
      A     #Rapper.auto_mode_control;
      AN    M 9.5;
      =     #Rapper.man_mode_locked;
      CALL  FC 21 (
           in_Ventil_Typ            := 0,
           in_Handbedienung_erlaubt := TRUE,
           in_Quitt_Stoerung_noetig := FALSE,
           in_Quitt_Stoerung        := TRUE,
           in_Anlage_ein            := #I_xSystemActive,
           in_Ansteuerung_Ventil    := #Rapper.auto_mode_control,
           in_Eingang_angesteuert   := FALSE,
           in_Eingang_nicht_angest  := FALSE,
           io_Ausgang_Ventil        := #q_xRepperValve,
           io_Ventil_in_Betrieb     := #Rapper.valve_in_operation,
           io_Stoerung              := #Rapper.fault,
           io_Ventilstruktur        := #Rapper);	// no feedback
NETWORK
TITLE = ------------------HOPPER'S STATES(REC/HP)-----------------------
NETWORK
TITLE = Intern statuses(full, filled, empty)
      A     #INTERNAL.Switches.xHighLevelCovered;
      =     #INTERNAL.ReceiverStatus.xFull;
//filled
      A     #SEQUENCES.Filling.RELEASE;
      A     #AngleValve.valve_in_operation;
      O     #INTERNAL.ReceiverStatus.xFull;
      S     #INTERNAL.ReceiverStatus.xFilled;
      A     #SEQUENCES.Discharging.RELEASE;
      A(;
      A     #TIMERS.TON_DischargingTime.Q;
      A     #INTERNAL.ProcessStatus.xRequestPM;
      O;
      A     #INTERNAL.Switches.xPendulumFlapClosed;
      );
      AN    #INTERNAL.ReceiverStatus.xFull;
      O;
      A     #HMI.CMD.xSetEmpty;	// from VISU
      AN    #INTERNAL.ReceiverStatus.xFull;
      AN    #SEQUENCES.Filling.ACTIVE;
      AN    #SEQUENCES.Filling.CLEANING;
      R     #INTERNAL.ReceiverStatus.xFilled;
//empty
      AN    #INTERNAL.ReceiverStatus.xFilled;
      =     #INTERNAL.ReceiverStatus.xEmpty;
NETWORK
TITLE = -------------------LAMPS/TASTER LIGHTS--------------------------
NETWORK
TITLE = Traffic Lamps
// red 
      A     #SEQUENCES.Discharging.FAULTED;
      O     #SEQUENCES.Filling.FAULTED;
      =     #INTERNAL.BUTTONS_LAMPS.Red.Steady;
      A     #fNotEnoughMaterial;
      =     #INTERNAL.BUTTONS_LAMPS.Red.Flash;
      CLR;
      =     #INTERNAL.BUTTONS_LAMPS.Red.DoubleFlash;
      CALL  FC 25 (
           Steady                   := #INTERNAL.BUTTONS_LAMPS.Red.Steady,
           Flash                    := #INTERNAL.BUTTONS_LAMPS.Red.Flash,
           DoubleFlash              := #INTERNAL.BUTTONS_LAMPS.Red.DoubleFlash,
           LampTest                 := M 9.7,
           Lamp                     := #q_xRedLamp);
//yellow
      A     #IF_VP.STATUS.STATE.xPressureFault;
      =     #INTERNAL.BUTTONS_LAMPS.Yellow.Steady;
      A     #HMI.STATE.xFull;
      =     #INTERNAL.BUTTONS_LAMPS.Yellow.Flash;
      A     #SEQUENCES.Filling.CLEANING;
      =     #INTERNAL.BUTTONS_LAMPS.Yellow.DoubleFlash;
      CALL  FC 25 (
           Steady                   := #INTERNAL.BUTTONS_LAMPS.Yellow.Steady,
           Flash                    := #INTERNAL.BUTTONS_LAMPS.Yellow.Flash,
           DoubleFlash              := #INTERNAL.BUTTONS_LAMPS.Yellow.DoubleFlash,
           LampTest                 := M 9.7,
           Lamp                     := #q_xYellowLamp);
//green
      AN    #SEQUENCES.Discharging.FAULTED;
      AN    #SEQUENCES.Filling.FAULTED;
      =     #INTERNAL.BUTTONS_LAMPS.Green.Steady;
      A     #SEQUENCES.Discharging.ACTIVE;
      A     #SEQUENCES.Filling.ACTIVE;
      =     #INTERNAL.BUTTONS_LAMPS.Green.Flash;
      CLR;
      =     #INTERNAL.BUTTONS_LAMPS.Green.DoubleFlash;
      CALL  FC 25 (
           Steady                   := #INTERNAL.BUTTONS_LAMPS.Green.Steady,
           Flash                    := #INTERNAL.BUTTONS_LAMPS.Green.Flash,
           DoubleFlash              := #INTERNAL.BUTTONS_LAMPS.Green.DoubleFlash,
           LampTest                 := M 9.7,
           Lamp                     := #q_xGreenLamp);
NETWORK
TITLE = Discharging: FAULTED to STORAGE
      O     #f_xFullReceiver;
      O     #f_xNoStartConditions;
      =     #SEQUENCES.Discharging.FAULTED;
NETWORK
TITLE = ----------------------OUTPUT PFCs-------------------------------
NETWORK
TITLE = -------------------------STATUSES HMI---------------------------
NETWORK
TITLE = -----------------------INTERFACES-------------------------------
NETWORK
TITLE = Storage location
      L     #I_iIFStorageDB;
      T     #INTERNAL.IF.Storage.StorageLocation_DB;
      L     #I_iIFStorageDW;
      T     #INTERNAL.IF.Storage.StorageLocation_DW;
      SET;
      =     #IF_Storage.CONTROL.CMD.xConnect;
      CALL  FC 40 (
           i_Freigabe               := #IF_Storage.CONTROL.CMD.xConnect,
           i_Ziel_DB                := #INTERNAL.IF.Storage.StorageLocation_DB,
           i_Ziel_DW                := #INTERNAL.IF.Storage.StorageLocation_DW,
           i_SST_von_Ziel           := #IF_Storage.STATUS,
           i_SST_an_Ziel            := #IF_Storage.CONTROL,
           Ziel_frei                := #INTERNAL.IF.Storage.IF_Silo_free);
      NOP   0;
NETWORK
TITLE = Blower
      L     #I_iIFVacuumPumpDB;
      T     #INTERNAL.IF.Blower.Blower_DB;
      L     #I_iIFVacuumPumpDW;
      T     #INTERNAL.IF.Blower.Blower_DW;
      CALL  FC 40 (
           i_Freigabe               := #IF_VP.CONTROL.CMD.xRequest,
           i_Ziel_DB                := #INTERNAL.IF.Blower.Blower_DB,
           i_Ziel_DW                := #INTERNAL.IF.Blower.Blower_DW,
           i_SST_von_Ziel           := #IF_VP.STATUS,
           i_SST_an_Ziel            := #IF_VP.CONTROL,
           Ziel_frei                := #INTERNAL.IF.Blower.Blower_free);
END_FUNCTION_BLOCK

